LIN {X -192.412,Y -0.639,Z -49.375,A 0.015,B 0.000,C 180.000} C_DIS
LIN {X -191.183,Y 5.850,Z -49.619,A 0.015,B 0.000,C 180.000} C_DIS
LIN {X -196.636,Y 9.577,Z -49.863,A 0.015,B 0.000,C 180.000} C_DIS
LIN {X -202.235,Y 6.074,Z -50.107,A 0.015,B 0.000,C 180.000} C_DIS
LIN {X -201.270,Y -0.459,Z -50.351,A 0.015,B 0.000,C 180.000} C_DIS
LIN {X -194.897,Y -2.193,Z -50.595,A 0.015,B 0.000,C -180.000} C_DIS
LIN {X -190.755,Y 2.951,Z -50.839,A 0.015,B 0.000,C 180.000} C_DIS
LIN {X -193.808,Y 8.807,Z -51.083,A 0.015,B 0.000,C 180.000} C_DIS
LIN {X -200.397,Y 8.357,Z -51.327,A 0.015,B 0.000,C -180.000} C_DIS
LIN {X -202.624,Y 2.139,Z -51.571,A 0.015,B 0.000,C -180.000} C_DIS
LIN {X -197.821,Y -2.393,Z -51.815,A 0.015,B 0.000,C 180.000} C_DIS
LIN {X -191.743,Y 0.192,Z -52.060,A 0.015,B 0.000,C -180.000} C_DIS
LIN {X -191.677,Y 6.796,Z -52.304,A 0.015,B 0.000,C 180.000} C_DIS
LIN {X -197.700,Y 9.504,Z -52.548,A 0.015,B -0.000,C 180.000} C_DIS
LIN {X -202.595,Y 5.070,Z -52.792,A 0.015,B 0.000,C 180.000} C_DIS
LIN {X -200.494,Y -1.191,Z -53.036,A 0.015,B 0.000,C 180.000} C_DIS
LIN {X -193.915,Y -1.775,Z -53.280,A 0.015,B 0.000,C -180.000} C_DIS
LIN {X -190.744,Y 4.018,Z -53.524,A 0.015,B -0.000,C 180.000} C_DIS
LIN {X -194.781,Y 9.245,Z -53.768,A 0.015,B 0.000,C -180.000} C_DIS
LIN {X -201.188,Y 7.640,Z -54.012,A 0.015,B 0.000,C -180.000} C_DIS
LIN {X -202.285,Y 1.128,Z -54.256,A 0.015,B -0.000,C 180.000} C_DIS
LIN {X -196.758,Y -2.487,Z -54.500,A 0.015,B 0.000,C 180.000} C_DIS
LIN {X -193.305,Y -2.487,Z -54.500,A 0.015,B 0.000,C 180.000} C_DIS
CIRC {X -191.945,Y -1.389,Z -54.500,A 0.015,B 0.000,C 180.000},{X -192.732,Y 0.173,Z -54.500,A 0.015,B 0.000,C 180.000} C_DIS
CIRC {X -193.494,Y 0.521,Z -54.500,A 0.015,B 0.000,C -180.000},{X -194.253,Y 0.875,Z -54.500,A 0.015,B -0.000,C -180.000} C_DIS
CIRC {X -195.005,Y 1.244,Z -54.500,A 0.015,B 0.000,C 180.000},{X -195.745,Y 1.635,Z -54.500,A 0.015,B 0.000,C 180.000} C_DIS
CIRC {X -196.775,Y 1.894,Z -54.500,A 0.015,B 0.000,C -180.000},{X -197.801,Y 1.619,Z -54.500,A 0.015,B 0.000,C 180.000} C_DIS
CIRC {X -198.507,Y 1.231,Z -54.500,A 0.015,B 0.000,C -180.000},{X -199.224,Y 0.863,Z -54.500,A 0.015,B 0.000,C 180.000} C_DIS
CIRC {X -199.949,Y 0.511,Z -54.500,A 0.015,B 0.000,C 180.000},{X -200.680,Y 0.172,Z -54.500,A 0.015,B 0.000,C -180.000} C_DIS
CIRC {X -201.468,Y -1.389,Z -54.500,A 0.015,B -0.000,C 180.000},{X -200.108,Y -2.487,Z -54.500,A 0.015,B 0.000,C 180.000} C_DIS
LIN {X -196.758,Y -2.487,Z -54.500,A 0.015,B 0.000,C 180.000} C_DIS
CIRC {X -194.703,Y -3.109,Z -54.500,A 0.015,B -0.000,C 180.000},{X -193.339,Y -4.767,Z -54.500,A 0.015,B 0.000,C -180.000} C_DIS
CIRC {X -191.974,Y -6.424,Z -54.500,A 0.015,B 0.000,C -180.000},{X -189.919,Y -7.047,Z -54.500,A 0.015,B 0.000,C -180.000} C_DIS
LIN {X -172.141,Y -7.047,Z -54.500,A 0.015,B 0.000,C 180.000} C_DIS
CIRC {X -170.781,Y -5.948,Z -54.500,A 0.015,B -0.000,C -180.000},{X -171.568,Y -4.387,Z -54.500,A 0.015,B -0.000,C 180.000} C_DIS
CIRC {X -177.271,Y -1.878,Z -54.500,A 0.015,B -0.000,C -180.000},{X -183.023,Y 0.518,Z -54.500,A 0.015,B 0.000,C 180.000} C_DIS
CIRC {X -188.715,Y 3.061,Z -54.500,A 0.015,B 0.000,C 180.000},{X -194.211,Y 6.003,Z -54.500,A 0.015,B 0.000,C 180.000} C_DIS
CIRC {X -196.812,Y 6.694,Z -54.500,A 0.015,B 0.000,C -180.000},{X -199.402,Y 5.963,Z -54.500,A 0.015,B -0.000,C -180.000} C_DIS
CIRC {X -204.829,Y 2.985,Z -54.500,A 0.015,B 0.000,C -180.000},{X -210.480,Y 0.455,Z -54.500,A 0.015,B 0.000,C 180.000} C_DIS
CIRC {X -216.198,Y -1.904,Z -54.500,A 0.015,B 0.000,C 180.000},{X -221.864,Y -4.387,Z -54.500,A 0.015,B -0.000,C 180.000} C_DIS
CIRC {X -222.652,Y -5.948,Z -54.500,A 0.015,B 0.000,C -180.000},{X -221.292,Y -7.047,Z -54.500,A 0.015,B 0.000,C 180.000} C_DIS
LIN {X -189.919,Y -7.047,Z -54.500,A 0.015,B 0.000,C -180.000} C_DIS
CIRC {X -187.085,Y -7.904,Z -54.500,A 0.015,B 0.000,C 180.000},{X -185.204,Y -10.190,Z -54.500,A 0.015,B -0.000,C -180.000} C_DIS
CIRC {X -183.322,Y -12.476,Z -54.500,A 0.015,B 0.000,C -180.000},{X -180.488,Y -13.334,Z -54.500,A 0.015,B 0.000,C 180.000} C_DIS
LIN {X -142.956,Y -13.334,Z -54.500,A 0.015,B 0.000,C 180.000} C_DIS
CIRC {X -141.596,Y -12.235,Z -54.500,A 0.015,B 0.000,C 180.000},{X -142.383,Y -10.674,Z -54.500,A 0.015,B 0.000,C 180.000} C_DIS
LIN {X -189.172,Y 10.284,Z -54.500,A 0.015,B -0.000,C 180.000} C_DIS
CIRC {X -190.364,Y 10.896,Z -54.500,A 0.015,B 0.000,C 180.000},{X -191.488,Y 11.625,Z -54.500,A 0.015,B 0.000,C -180.000} C_DIS
CIRC {X -192.572,Y 12.410,Z -54.500,A 0.015,B 0.000,C 180.000},{X -193.651,Y 13.201,Z -54.500,A 0.015,B 0.000,C 180.000} C_DIS
CIRC {X -196.677,Y 14.214,Z -54.500,A 0.015,B 0.000,C 180.000},{X -199.724,Y 13.268,Z -54.500,A 0.015,B 0.000,C -180.000} C_DIS
CIRC {X -200.958,Y 12.395,Z -54.500,A 0.015,B 0.000,C 180.000},{X -202.187,Y 11.516,Z -54.500,A 0.015,B 0.000,C -180.000} C_DIS
CIRC {X -203.459,Y 10.695,Z -54.500,A 0.015,B 0.000,C -180.000},{X -204.805,Y 10.005,Z -54.500,A 0.015,B 0.000,C -180.000} C_DIS
LIN {X -251.078,Y -10.675,Z -54.500,A 0.015,B 0.000,C -180.000} C_DIS
CIRC {X -251.866,Y -12.235,Z -54.500,A 0.015,B 0.000,C 180.000},{X -250.505,Y -13.334,Z -54.500,A 0.015,B 0.000,C -180.000} C_DIS
LIN {X -180.488,Y -13.334,Z -54.500,A 0.015,B 0.000,C 180.000} C_DIS
CIRC {X -177.654,Y -14.192,Z -54.500,A 0.015,B 0.000,C 180.000},{X -175.772,Y -16.478,Z -54.500,A 0.015,B 0.000,C -180.000} C_DIS
CIRC {X -173.891,Y -18.763,Z -54.500,A 0.015,B -0.000,C -180.000},{X -171.057,Y -19.621,Z -54.500,A 0.015,B 0.000,C 180.000} C_DIS
LIN {X -113.771,Y -19.621,Z -54.500,A 0.015,B 0.000,C 180.000} C_DIS
CIRC {X -112.410,Y -18.523,Z -54.500,A 0.015,B 0.000,C 180.000},{X -113.198,Y -16.962,Z -54.500,A 0.015,B 0.000,C 180.000} C_DIS
LIN {X -186.653,Y 15.858,Z -54.500,A 0.015,B 0.000,C -180.000} C_DIS
CIRC {X -189.034,Y 17.198,Z -54.500,A 0.015,B 0.000,C 180.000},{X -191.144,Y 18.934,Z -54.500,A 0.015,B 0.000,C -180.000} C_DIS
CIRC {X -193.015,Y 20.912,Z -54.500,A 0.015,B 0.000,C -180.000},{X -194.736,Y 23.023,Z -54.500,A 0.015,B 0.000,C 180.000} C_DIS
CIRC {X -196.819,Y 24.035,Z -54.500,A 0.015,B 0.000,C 180.000},{X -198.863,Y 22.946,Z -54.500,A 0.015,B 0.000,C 180.000} C_DIS
CIRC {X -199.889,Y 21.563,Z -54.500,A 0.015,B -0.000,C 180.000},{X -200.992,Y 20.240,Z -54.500,A 0.015,B 0.000,C -180.000} C_DIS
CIRC {X -202.216,Y 19.026,Z -54.500,A 0.015,B 0.000,C 180.000},{X -203.590,Y 17.983,Z -54.500,A 0.015,B 0.000,C 180.000} C_DIS
CIRC {X -204.508,Y 17.359,Z -54.500,A 0.015,B -0.000,C -180.000},{X -205.410,Y 16.710,Z -54.500,A 0.015,B 0.000,C 180.000} C_DIS
CIRC {X -206.337,Y 16.098,Z -54.500,A 0.015,B 0.000,C -180.000},{X -207.325,Y 15.587,Z -54.500,A 0.015,B 0.000,C 180.000} C_DIS
LIN {X -280.291,Y -16.962,Z -54.500,A 0.015,B 0.000,C -180.000} C_DIS
CIRC {X -281.079,Y -18.523,Z -54.500,A 0.015,B 0.000,C 180.000},{X -279.719,Y -19.621,Z -54.500,A 0.015,B -0.000,C -180.000} C_DIS
LIN {X -171.057,Y -19.621,Z -54.500,A 0.015,B -0.000,C 180.000} C_DIS
LIN {X -170.448,Y -19.466,Z -54.330,A 0.015,B 0.000,C 180.000} C_DIS
LIN {X -170.089,Y -19.174,Z -53.865,A 0.015,B 0.000,C 180.000} C_DIS
LIN {X -169.988,Y -19.038,Z -53.230,A 0.015,B 0.000,C 180.000} C_DIS
$VEL.CP = 1.00000
LIN {X -169.988,Y -19.038,Z 11.000,A 0.015,B 0.000,C -180.000} C_DIS
$VEL.CP = 1.00000
LIN {X -57.220,Y 262.988,Z 11.000,A 0.015,B -0.000,C -180.000} C_DIS
$VEL.CP = 1.00000
LIN {X -57.220,Y 262.988,Z -32.731,A 0.015,B 0.000,C 180.000} C_DIS
$VEL.CP = 0.10000
LIN {X -57.218,Y 263.151,Z -33.353,A 0.015,B 0.000,C 180.000} C_DIS
LIN {X -57.234,Y 263.597,Z -33.816,A 0.015,B 0.000,C -180.000} C_DIS
LIN {X -57.310,Y 264.209,Z -34.000,A 0.015,B 0.000,C -180.000} C_DIS
LIN {X -61.835,Y 269.020,Z -34.244,A 0.015,B 0.000,C 180.000} C_DIS
LIN {X -68.056,Y 266.803,Z -34.488,A 0.015,B -0.000,C -180.000} C_DIS
LIN {X -68.517,Y 260.215,Z -34.732,A 0.015,B -0.000,C -180.000} C_DIS
LIN {X -62.666,Y 257.152,Z -34.976,A 0.015,B 0.000,C 180.000} C_DIS
LIN {X -57.515,Y 261.285,Z -35.220,A 0.015,B 0.000,C -180.000} C_DIS
LIN {X -59.238,Y 267.661,Z -35.464,A 0.015,B 0.000,C -180.000} C_DIS
LIN {X -65.770,Y 268.637,Z -35.708,A 0.015,B 0.000,C -180.000} C_DIS
LIN {X -69.282,Y 263.044,Z -35.952,A 0.015,B 0.000,C -180.000} C_DIS
LIN {X -65.565,Y 257.585,Z -36.196,A 0.015,B -0.000,C 180.000} C_DIS
LIN {X -59.074,Y 258.803,Z -36.440,A 0.015,B 0.000,C -180.000} C_DIS
LIN {X -57.589,Y 265.238,Z -36.685,A 0.015,B 0.000,C -180.000} C_DIS
LIN {X -62.890,Y 269.178,Z -36.929,A 0.015,B -0.000,C 180.000} C_DIS
LIN {X -68.623,Y 265.900,Z -37.173,A 0.015,B -0.000,C 180.000} C_DIS
LIN {X -67.917,Y 259.333,Z -37.417,A 0.015,B 0.000,C 180.000} C_DIS
LIN {X -61.618,Y 257.348,Z -37.661,A 0.015,B 0.000,C -180.000} C_DIS
LIN {X -57.275,Y 262.324,Z -37.905,A 0.015,B 0.000,C -180.000} C_DIS
LIN {X -60.094,Y 268.297,Z -38.149,A 0.015,B 0.000,C 180.000} C_DIS
LIN {X -66.696,Y 268.108,Z -38.393,A 0.015,B 0.000,C 180.000} C_DIS
LIN {X -69.168,Y 261.983,Z -38.637,A 0.015,B 0.000,C -180.000} C_DIS
LIN {X -64.547,Y 257.264,Z -38.881,A 0.015,B 0.000,C -180.000} C_DIS
LIN {X -58.372,Y 259.607,Z -39.125,A 0.015,B 0.000,C 180.000} C_DIS
LIN {X -58.044,Y 266.203,Z -39.369,A 0.015,B 0.000,C 180.000} C_DIS
LIN {X -63.956,Y 269.147,Z -39.613,A 0.015,B 0.000,C -180.000} C_DIS
LIN {X -69.022,Y 264.910,Z -39.857,A 0.015,B 0.000,C 180.000} C_DIS
LIN {X -67.171,Y 258.571,Z -40.101,A 0.015,B -0.000,C 180.000} C_DIS
LIN {X -60.621,Y 257.727,Z -40.345,A 0.015,B 0.000,C -180.000} C_DIS
LIN {X -57.222,Y 263.390,Z -40.589,A 0.015,B 0.000,C 180.000} C_DIS
LIN {X -61.049,Y 268.772,Z -40.833,A 0.015,B 0.000,C -180.000} C_DIS
LIN {X -67.514,Y 267.423,Z -41.077,A 0.015,B 0.000,C -180.000} C_DIS
LIN {X -68.869,Y 260.959,Z -41.321,A 0.015,B 0.000,C -180.000} C_DIS
LIN {X -63.489,Y 257.128,Z -41.565,A 0.015,B 0.000,C 180.000} C_DIS
LIN {X -57.824,Y 260.521,Z -41.810,A 0.015,B 0.000,C 180.000} C_DIS
LIN {X -58.662,Y 267.072,Z -42.054,A 0.015,B 0.000,C 180.000} C_DIS
LIN {X -65.000,Y 268.929,Z -42.298,A 0.015,B 0.000,C -180.000} C_DIS
LIN {X -69.241,Y 263.866,Z -42.542,A 0.015,B 0.000,C 180.000} C_DIS
LIN {X -66.302,Y 257.952,Z -42.786,A 0.015,B 0.000,C 180.000} C_DIS
LIN {X -59.705,Y 258.275,Z -43.030,A 0.015,B 0.000,C 180.000} C_DIS
LIN {X -57.358,Y 264.448,Z -43.274,A 0.015,B 0.000,C -180.000} C_DIS
LIN {X -62.073,Y 269.072,Z -43.518,A 0.015,B 0.000,C -180.000} C_DIS
LIN {X -68.199,Y 266.606,Z -43.762,A 0.015,B 0.000,C -180.000} C_DIS
LIN {X -68.394,Y 260.004,Z -44.006,A 0.015,B 0.000,C 180.000} C_DIS
LIN {X -62.424,Y 257.180,Z -44.250,A 0.015,B 0.000,C -180.000} C_DIS
LIN {X -57.444,Y 261.518,Z -44.494,A 0.015,B 0.000,C 180.000} C_DIS
LIN {X -59.424,Y 267.819,Z -44.738,A 0.015,B 0.000,C -180.000} C_DIS
LIN {X -65.989,Y 268.531,Z -44.982,A 0.015,B 0.000,C -180.000} C_DIS
LIN {X -69.272,Y 262.800,Z -45.226,A 0.015,B 0.000,C 180.000} C_DIS
LIN {X -65.338,Y 257.496,Z -45.470,A 0.015,B -0.000,C 180.000} C_DIS
LIN {X -58.901,Y 258.976,Z -45.714,A 0.015,B -0.000,C 180.000} C_DIS
LIN {X -57.678,Y 265.465,Z -45.958,A 0.015,B 0.000,C -180.000} C_DIS
LIN {X -63.133,Y 269.187,Z -46.202,A 0.015,B -0.000,C 180.000} C_DIS
LIN {X -68.729,Y 265.680,Z -46.446,A 0.015,B 0.000,C 180.000} C_DIS
LIN {X -67.759,Y 259.148,Z -46.690,A 0.015,B 0.000,C -180.000} C_DIS
LIN {X -61.384,Y 257.419,Z -46.935,A 0.015,B -0.000,C -180.000} C_DIS
LIN {X -57.247,Y 262.567,Z -47.179,A 0.015,B 0.000,C 180.000} C_DIS
LIN {X -60.305,Y 268.420,Z -47.423,A 0.015,B 0.000,C -180.000} C_DIS
LIN {X -66.893,Y 267.964,Z -47.667,A 0.015,B 0.000,C -180.000} C_DIS
LIN {X -69.116,Y 261.745,Z -47.911,A 0.015,B 0.000,C 180.000} C_DIS
LIN {X -64.308,Y 257.217,Z -48.155,A 0.015,B -0.000,C 180.000} C_DIS
LIN {X -58.233,Y 259.807,Z -48.399,A 0.015,B -0.000,C 180.000} C_DIS
LIN {X -58.171,Y 266.411,Z -48.643,A 0.015,B 0.000,C 180.000} C_DIS
LIN {X -64.197,Y 269.114,Z -48.887,A 0.015,B 0.000,C -180.000} C_DIS
LIN {X -69.088,Y 264.676,Z -49.131,A 0.015,B -0.000,C -180.000} C_DIS
LIN {X -66.982,Y 258.416,Z -49.375,A 0.015,B 0.000,C 180.000} C_DIS
LIN {X -60.403,Y 257.838,Z -49.619,A 0.015,B 0.000,C 180.000} C_DIS
LIN {X -57.237,Y 263.633,Z -49.863,A 0.015,B 0.000,C 180.000} C_DIS
LIN {X -61.278,Y 268.857,Z -50.107,A 0.015,B 0.000,C 180.000} C_DIS
LIN {X -67.683,Y 267.247,Z -50.351,A 0.015,B 0.000,C -180.000} C_DIS
LIN {X -68.775,Y 260.734,Z -50.595,A 0.015,B 0.000,C 180.000} C_DIS
LIN {X -63.246,Y 257.123,Z -50.839,A 0.015,B 0.000,C -180.000} C_DIS
LIN {X -57.721,Y 260.743,Z -51.083,A 0.015,B 0.000,C -180.000} C_DIS
LIN {X -58.824,Y 267.255,Z -51.327,A 0.015,B -0.000,C 180.000} C_DIS
LIN {X -65.232,Y 268.854,Z -51.571,A 0.015,B 0.000,C -180.000} C_DIS
LIN {X -69.265,Y 263.624,Z -51.815,A 0.015,B 0.000,C 180.000} C_DIS
LIN {X -66.089,Y 257.833,Z -52.060,A 0.015,B 0.000,C 180.000} C_DIS
LIN {X -59.511,Y 258.422,Z -52.304,A 0.015,B 0.000,C 180.000} C_DIS
LIN {X -57.415,Y 264.685,Z -52.548,A 0.015,B 0.000,C -180.000} C_DIS
LIN {X -62.313,Y 269.115,Z -52.792,A 0.015,B 0.000,C -180.000} C_DIS
LIN {X -68.335,Y 266.403,Z -53.036,A 0.015,B -0.000,C 180.000} C_DIS
LIN {X -68.262,Y 259.799,Z -53.280,A 0.015,B 0.000,C 180.000} C_DIS
LIN {X -62.183,Y 257.219,Z -53.524,A 0.015,B 0.000,C 180.000} C_DIS
LIN {X -57.383,Y 261.754,Z -53.768,A 0.015,B -0.000,C -180.000} C_DIS
LIN {X -59.615,Y 267.970,Z -54.012,A 0.015,B 0.000,C 180.000} C_DIS
LIN {X -66.204,Y 268.416,Z -54.256,A 0.015,B 0.000,C -180.000} C_DIS
LIN {X -69.253,Y 262.557,Z -54.500,A 0.015,B 0.000,C 180.000} C_DIS
LIN {X -65.146,Y 221.387,Z -54.500,A 0.015,B 0.000,C 180.000} C_DIS
CIRC {X -63.949,Y 220.356,Z -54.500,A 0.015,B 0.000,C -180.000},{X -62.860,Y 221.500,Z -54.500,A 0.015,B 0.000,C 180.000} C_DIS
LIN {X -62.861,Y 263.241,Z -54.500,A 0.015,B 0.000,C 180.000} C_DIS
CIRC {X -63.692,Y 265.248,Z -54.500,A 0.015,B -0.000,C -180.000},{X -65.699,Y 266.079,Z -54.500,A 0.015,B 0.000,C -180.000} C_DIS
LIN {X -66.469,Y 266.079,Z -54.500,A 0.015,B 0.000,C 180.000} C_DIS
CIRC {X -68.573,Y 265.145,Z -54.500,A 0.015,B 0.000,C 180.000},{X -69.293,Y 262.959,Z -54.500,A 0.015,B -0.000,C -180.000} C_DIS
LIN {X -69.253,Y 262.557,Z -54.500,A 0.015,B 0.000,C 180.000} C_DIS
CIRC {X -69.735,Y 260.112,Z -54.500,A 0.015,B 0.000,C -180.000},{X -71.492,Y 258.345,Z -54.500,A 0.015,B 0.000,C 180.000} C_DIS
CIRC {X -73.249,Y 256.577,Z -54.500,A 0.015,B 0.000,C -180.000},{X -73.731,Y 254.132,Z -54.500,A 0.015,B -0.000,C -180.000} C_DIS
LIN {X -66.932,Y 185.980,Z -54.500,A 0.015,B 0.000,C -180.000} C_DIS
CIRC {X -66.441,Y 184.456,Z -54.500,A 0.015,B 0.000,C 180.000},{X -65.366,Y 183.268,Z -54.500,A 0.015,B 0.000,C 180.000} C_DIS
LIN {X -60.809,Y 179.993,Z -54.500,A 0.015,B 0.000,C -180.000} C_DIS
CIRC {X -58.680,Y 179.834,Z -54.500,A 0.015,B 0.000,C -180.000},{X -57.566,Y 181.656,Z -54.500,A 0.015,B -0.000,C -180.000} C_DIS
LIN {X -57.569,Y 267.519,Z -54.500,A 0.015,B -0.000,C -180.000} C_DIS
CIRC {X -58.697,Y 270.243,Z -54.500,A 0.015,B 0.000,C 180.000},{X -61.422,Y 271.372,Z -54.500,A 0.015,B 0.000,C 180.000} C_DIS
LIN {X -71.668,Y 271.371,Z -54.500,A 0.015,B 0.000,C 180.000} C_DIS
CIRC {X -74.207,Y 270.245,Z -54.500,A 0.015,B 0.000,C 180.000},{X -75.076,Y 267.607,Z -54.500,A 0.015,B -0.000,C -180.000} C_DIS
LIN {X -73.731,Y 254.132,Z -54.500,A 0.015,B 0.000,C 180.000} C_DIS
CIRC {X -74.442,Y 250.524,Z -54.500,A 0.015,B 0.000,C -180.000},{X -77.035,Y 247.916,Z -54.500,A 0.015,B 0.000,C -180.000} C_DIS
CIRC {X -79.628,Y 245.308,Z -54.500,A 0.015,B 0.000,C -180.000},{X -80.339,Y 241.700,Z -54.500,A 0.015,B 0.000,C -180.000} C_DIS
LIN {X -74.727,Y 185.448,Z -54.500,A 0.015,B -0.000,C -180.000} C_DIS
CIRC {X -73.159,Y 180.577,Z -54.500,A 0.015,B 0.000,C 180.000},{X -69.725,Y 176.784,Z -54.500,A 0.015,B -0.000,C -180.000} C_DIS
LIN {X -52.999,Y 164.764,Z -54.500,A 0.015,B 0.000,C -180.000} C_DIS
CIRC {X -50.869,Y 164.604,Z -54.500,A 0.015,B -0.000,C -180.000},{X -49.756,Y 166.427,Z -54.500,A 0.015,B -0.000,C -180.000} C_DIS
LIN {X -49.759,Y 275.329,Z -54.500,A 0.015,B 0.000,C -180.000} C_DIS
CIRC {X -50.888,Y 278.053,Z -54.500,A 0.015,B 0.000,C 180.000},{X -53.612,Y 279.182,Z -54.500,A 0.015,B 0.000,C -180.000} C_DIS
LIN {X -80.296,Y 279.181,Z -54.500,A 0.015,B 0.000,C -180.000} C_DIS
CIRC {X -82.835,Y 278.055,Z -54.500,A 0.015,B 0.000,C 180.000},{X -83.703,Y 275.416,Z -54.500,A 0.015,B 0.000,C -180.000} C_DIS
LIN {X -80.339,Y 241.700,Z -54.500,A 0.015,B 0.000,C -180.000} C_DIS
CIRC {X -81.050,Y 238.092,Z -54.500,A 0.015,B -0.000,C 180.000},{X -83.644,Y 235.484,Z -54.500,A 0.015,B 0.000,C 180.000} C_DIS
CIRC {X -86.237,Y 232.876,Z -54.500,A 0.015,B 0.000,C 180.000},{X -86.948,Y 229.268,Z -54.500,A 0.015,B 0.000,C 180.000} C_DIS
LIN {X -82.181,Y 181.488,Z -54.500,A 0.015,B 0.000,C -180.000} C_DIS
CIRC {X -80.519,Y 176.328,Z -54.500,A 0.015,B -0.000,C -180.000},{X -76.882,Y 172.310,Z -54.500,A 0.015,B -0.000,C 180.000} C_DIS
LIN {X -45.189,Y 149.534,Z -54.500,A 0.015,B 0.000,C -180.000} C_DIS
CIRC {X -43.059,Y 149.375,Z -54.500,A 0.015,B -0.000,C 180.000},{X -41.946,Y 151.197,Z -54.500,A 0.015,B 0.000,C -180.000} C_DIS
LIN {X -41.949,Y 283.139,Z -54.500,A 0.015,B 0.000,C 180.000} C_DIS
CIRC {X -43.078,Y 285.863,Z -54.500,A 0.015,B 0.000,C -180.000},{X -45.802,Y 286.992,Z -54.500,A 0.015,B -0.000,C 180.000} C_DIS
LIN {X -88.923,Y 286.991,Z -54.500,A 0.015,B -0.000,C 180.000} C_DIS
CIRC {X -91.462,Y 285.864,Z -54.500,A 0.015,B 0.000,C 180.000},{X -92.331,Y 283.226,Z -54.500,A 0.015,B -0.000,C 180.000} C_DIS
LIN {X -86.948,Y 229.268,Z -54.500,A 0.015,B -0.000,C -180.000} C_DIS
CIRC {X -87.659,Y 225.660,Z -54.500,A 0.015,B 0.000,C -180.000},{X -90.252,Y 223.052,Z -54.500,A 0.015,B 0.000,C -180.000} C_DIS
CIRC {X -92.845,Y 220.444,Z -54.500,A 0.015,B 0.000,C 180.000},{X -93.556,Y 216.836,Z -54.500,A 0.015,B 0.000,C 180.000} C_DIS
LIN {X -89.602,Y 177.203,Z -54.500,A 0.015,B 0.000,C 180.000} C_DIS
CIRC {X -87.941,Y 172.044,Z -54.500,A 0.015,B 0.000,C 180.000},{X -84.303,Y 168.025,Z -54.500,A 0.015,B -0.000,C 180.000} C_DIS
LIN {X -37.378,Y 134.304,Z -54.500,A 0.015,B 0.000,C -180.000} C_DIS
CIRC {X -35.249,Y 134.145,Z -54.500,A 0.015,B 0.000,C 180.000},{X -34.136,Y 135.967,Z -54.500,A 0.015,B -0.000,C -180.000} C_DIS
LIN {X -34.140,Y 290.949,Z -54.500,A 0.015,B 0.000,C -180.000} C_DIS
CIRC {X -35.268,Y 293.673,Z -54.500,A 0.015,B 0.000,C 180.000},{X -37.993,Y 294.802,Z -54.500,A 0.015,B 0.000,C 180.000} C_DIS
LIN {X -97.551,Y 294.800,Z -54.500,A 0.015,B -0.000,C 180.000} C_DIS
CIRC {X -100.090,Y 293.674,Z -54.500,A 0.015,B -0.000,C 180.000},{X -100.959,Y 291.036,Z -54.500,A 0.015,B 0.000,C 180.000} C_DIS
LIN {X -93.556,Y 216.836,Z -54.500,A 0.015,B 0.000,C -180.000} C_DIS
CIRC {X -94.268,Y 213.222,Z -54.500,A 0.015,B 0.000,C -180.000},{X -96.864,Y 210.610,Z -54.500,A 0.015,B 0.000,C -180.000} C_DIS
CIRC {X -99.460,Y 207.998,Z -54.500,A 0.015,B 0.000,C -180.000},{X -100.171,Y 204.384,Z -54.500,A 0.015,B 0.000,C -180.000} C_DIS
LIN {X -97.023,Y 172.919,Z -54.500,A 0.015,B 0.000,C -180.000} C_DIS
CIRC {X -95.362,Y 167.760,Z -54.500,A 0.015,B 0.000,C -180.000},{X -91.724,Y 163.741,Z -54.500,A 0.015,B 0.000,C 180.000} C_DIS
LIN {X -29.568,Y 119.075,Z -54.500,A 0.015,B 0.000,C 180.000} C_DIS
CIRC {X -27.439,Y 118.915,Z -54.500,A 0.015,B 0.000,C -180.000},{X -26.325,Y 120.738,Z -54.500,A 0.015,B 0.000,C -180.000} C_DIS
LIN {X -26.330,Y 298.759,Z -54.500,A 0.015,B 0.000,C 180.000} C_DIS
CIRC {X -27.459,Y 301.483,Z -54.500,A 0.015,B -0.000,C 180.000},{X -30.183,Y 302.612,Z -54.500,A 0.015,B 0.000,C -180.000} C_DIS
LIN {X -106.248,Y 302.610,Z -54.500,A 0.015,B 0.000,C 180.000} C_DIS
CIRC {X -108.774,Y 301.483,Z -54.500,A 0.015,B 0.000,C 180.000},{X -109.624,Y 298.852,Z -54.500,A 0.015,B 0.000,C 180.000} C_DIS
LIN {X -100.171,Y 204.384,Z -54.500,A 0.015,B -0.000,C 180.000} C_DIS
CIRC {X -100.875,Y 200.830,Z -54.500,A 0.015,B 0.000,C -180.000},{X -103.439,Y 198.271,Z -54.500,A 0.015,B 0.000,C 180.000} C_DIS
CIRC {X -105.996,Y 195.708,Z -54.500,A 0.015,B 0.000,C 180.000},{X -106.706,Y 192.157,Z -54.500,A 0.015,B 0.000,C -180.000} C_DIS
LIN {X -104.355,Y 167.741,Z -54.500,A 0.015,B 0.000,C -180.000} C_DIS
CIRC {X -102.950,Y 163.379,Z -54.500,A 0.015,B 0.000,C -180.000},{X -99.875,Y 159.981,Z -54.500,A 0.015,B -0.000,C -180.000} C_DIS
LIN {X -21.758,Y 103.845,Z -54.500,A 0.015,B -0.000,C 180.000} C_DIS
CIRC {X -19.628,Y 103.686,Z -54.500,A 0.015,B 0.000,C -180.000},{X -18.515,Y 105.508,Z -54.500,A 0.015,B 0.000,C 180.000} C_DIS
LIN {X -18.521,Y 306.569,Z -54.500,A 0.015,B 0.000,C 180.000} C_DIS
CIRC {X -19.649,Y 309.293,Z -54.500,A 0.015,B 0.000,C 180.000},{X -22.374,Y 310.422,Z -54.500,A 0.015,B 0.000,C -180.000} C_DIS
LIN {X -115.486,Y 310.419,Z -54.500,A 0.015,B -0.000,C 180.000} C_DIS
CIRC {X -117.830,Y 309.310,Z -54.500,A 0.015,B 0.000,C 180.000},{X -118.460,Y 306.795,Z -54.500,A 0.015,B -0.000,C -180.000} C_DIS
CIRC {X -117.276,Y 299.976,Z -54.500,A 0.015,B 0.000,C 180.000},{X -116.428,Y 293.107,Z -54.500,A 0.015,B 0.000,C -180.000} C_DIS
LIN {X -106.706,Y 192.157,Z -54.500,A 0.015,B -0.000,C -180.000} C_DIS
CIRC {X -107.419,Y 188.605,Z -54.500,A 0.015,B 0.000,C 180.000},{X -109.983,Y 186.044,Z -54.500,A 0.015,B 0.000,C -180.000} C_DIS
CIRC {X -112.546,Y 183.483,Z -54.500,A 0.015,B 0.000,C 180.000},{X -113.259,Y 179.930,Z -54.500,A 0.015,B 0.000,C 180.000} C_DIS
LIN {X -111.900,Y 165.827,Z -54.500,A 0.015,B -0.000,C 180.000} C_DIS
CIRC {X -111.841,Y 164.928,Z -54.500,A 0.015,B 0.000,C 180.000},{X -111.843,Y 164.026,Z -54.500,A 0.015,B 0.000,C 180.000} C_DIS
CIRC {X -111.879,Y 163.126,Z -54.500,A 0.015,B 0.000,C 180.000},{X -111.919,Y 162.226,Z -54.500,A 0.015,B 0.000,C 180.000} C_DIS
CIRC {X -111.054,Y 158.666,Z -54.500,A 0.015,B 0.000,C 180.000},{X -108.395,Y 156.145,Z -54.500,A 0.015,B 0.000,C 180.000} C_DIS
CIRC {X -107.575,Y 155.723,Z -54.500,A 0.015,B 0.000,C 180.000},{X -106.758,Y 155.295,Z -54.500,A 0.015,B 0.000,C 180.000} C_DIS
CIRC {X -105.958,Y 154.837,Z -54.500,A 0.015,B -0.000,C 180.000},{X -105.190,Y 154.325,Z -54.500,A 0.015,B 0.000,C 180.000} C_DIS
LIN {X -13.948,Y 88.615,Z -54.500,A 0.015,B 0.000,C -180.000} C_DIS
CIRC {X -11.818,Y 88.456,Z -54.500,A 0.015,B 0.000,C -180.000},{X -10.705,Y 90.278,Z -54.500,A 0.015,B 0.000,C 180.000} C_DIS
LIN {X -10.711,Y 314.379,Z -54.500,A 0.015,B 0.000,C 180.000} C_DIS
CIRC {X -11.840,Y 317.103,Z -54.500,A 0.015,B 0.000,C -180.000},{X -14.564,Y 318.232,Z -54.500,A 0.015,B -0.000,C 180.000} C_DIS
LIN {X -125.780,Y 318.229,Z -54.500,A 0.015,B -0.000,C -180.000} C_DIS
CIRC {X -127.944,Y 317.152,Z -54.500,A 0.015,B 0.000,C 180.000},{X -128.390,Y 314.776,Z -54.500,A 0.015,B -0.000,C 180.000} C_DIS
CIRC {X -125.771,Y 303.744,Z -54.500,A 0.015,B 0.000,C 180.000},{X -124.108,Y 292.528,Z -54.500,A 0.015,B -0.000,C 180.000} C_DIS
LIN {X -113.259,Y 179.930,Z -54.500,A 0.015,B -0.000,C 180.000} C_DIS
CIRC {X -113.965,Y 176.402,Z -54.500,A 0.015,B 0.000,C -180.000},{X -116.506,Y 173.856,Z -54.500,A 0.015,B -0.000,C -180.000} C_DIS
CIRC {X -119.051,Y 171.310,Z -54.500,A 0.015,B -0.000,C -180.000},{X -119.754,Y 167.781,Z -54.500,A 0.015,B -0.000,C 180.000} C_DIS
LIN {X -119.489,Y 165.070,Z -54.500,A 0.015,B 0.000,C 180.000} C_DIS
CIRC {X -119.427,Y 162.680,Z -54.500,A 0.015,B -0.000,C 180.000},{X -119.716,Y 160.306,Z -54.500,A 0.015,B -0.000,C -180.000} C_DIS
CIRC {X -120.244,Y 157.979,Z -54.500,A 0.015,B -0.000,C 180.000},{X -120.905,Y 155.686,Z -54.500,A 0.015,B 0.000,C -180.000} C_DIS
CIRC {X -120.644,Y 153.191,Z -54.500,A 0.015,B 0.000,C -180.000},{X -118.634,Y 151.690,Z -54.500,A 0.015,B 0.000,C 180.000} C_DIS
CIRC {X -116.926,Y 151.259,Z -54.500,A 0.015,B 0.000,C -180.000},{X -115.236,Y 150.764,Z -54.500,A 0.015,B 0.000,C -180.000} C_DIS
CIRC {X -113.576,Y 150.171,Z -54.500,A 0.015,B 0.000,C -180.000},{X -111.970,Y 149.447,Z -54.500,A 0.015,B 0.000,C 180.000} C_DIS
CIRC {X -111.373,Y 149.145,Z -54.500,A 0.015,B 0.000,C -180.000},{X -110.778,Y 148.837,Z -54.500,A 0.015,B 0.000,C 180.000} C_DIS
CIRC {X -110.196,Y 148.505,Z -54.500,A 0.015,B 0.000,C -180.000},{X -109.639,Y 148.134,Z -54.500,A 0.015,B 0.000,C 180.000} C_DIS
LIN {X -6.138,Y 73.385,Z -54.500,A 0.015,B 0.000,C -180.000} C_DIS
CIRC {X -4.008,Y 73.226,Z -54.500,A 0.015,B 0.000,C 180.000},{X -2.895,Y 75.048,Z -54.500,A 0.015,B -0.000,C -180.000} C_DIS
LIN {X -2.901,Y 322.189,Z -54.500,A 0.015,B -0.000,C -180.000} C_DIS
CIRC {X -4.030,Y 324.913,Z -54.500,A 0.015,B 0.000,C 180.000},{X -6.755,Y 326.042,Z -54.500,A 0.015,B 0.000,C -180.000} C_DIS
LIN {X -138.556,Y 326.038,Z -54.500,A 0.015,B 0.000,C -180.000} C_DIS
CIRC {X -140.500,Y 324.922,Z -54.500,A 0.015,B 0.000,C -180.000},{X -140.515,Y 322.681,Z -54.500,A 0.015,B 0.000,C 180.000} C_DIS
CIRC {X -138.936,Y 319.901,Z -54.500,A 0.015,B 0.000,C 180.000},{X -137.343,Y 317.129,Z -54.500,A 0.015,B 0.000,C -180.000} C_DIS
CIRC {X -135.984,Y 314.222,Z -54.500,A 0.015,B 0.000,C -180.000},{X -135.146,Y 311.124,Z -54.500,A 0.015,B 0.000,C -180.000} C_DIS
CIRC {X -134.260,Y 306.277,Z -54.500,A 0.015,B 0.000,C 180.000},{X -133.339,Y 301.438,Z -54.500,A 0.015,B 0.000,C 180.000} C_DIS
CIRC {X -132.503,Y 296.582,Z -54.500,A 0.015,B 0.000,C -180.000},{X -131.874,Y 291.695,Z -54.500,A 0.015,B 0.000,C 180.000} C_DIS
LIN {X -119.754,Y 167.781,Z -54.500,A 0.015,B 0.000,C -180.000} C_DIS
CIRC {X -120.533,Y 163.962,Z -54.500,A 0.015,B -0.000,C 180.000},{X -123.324,Y 161.243,Z -54.500,A 0.015,B 0.000,C 180.000} C_DIS
CIRC {X -126.370,Y 159.021,Z -54.500,A 0.015,B 0.000,C -180.000},{X -128.586,Y 155.970,Z -54.500,A 0.015,B 0.000,C -180.000} C_DIS
CIRC {X -129.163,Y 154.939,Z -54.500,A 0.015,B 0.000,C -180.000},{X -129.820,Y 153.956,Z -54.500,A 0.015,B 0.000,C 180.000} C_DIS
CIRC {X -133.257,Y 149.818,Z -54.500,A 0.015,B 0.000,C -180.000},{X -137.197,Y 146.156,Z -54.500,A 0.015,B 0.000,C 180.000} C_DIS
CIRC {X -137.836,Y 145.658,Z -54.500,A 0.015,B 0.000,C 180.000},{X -138.496,Y 145.188,Z -54.500,A 0.015,B -0.000,C -180.000} C_DIS
CIRC {X -139.174,Y 144.745,Z -54.500,A 0.015,B 0.000,C -180.000},{X -139.868,Y 144.327,Z -54.500,A 0.015,B 0.000,C 180.000} C_DIS
LIN {X -176.147,Y 123.347,Z -54.500,A 0.015,B 0.000,C -180.000} C_DIS
CIRC {X -181.598,Y 121.768,Z -54.500,A 0.015,B 0.000,C -180.000},{X -187.157,Y 122.914,Z -54.500,A 0.015,B 0.000,C 180.000} C_DIS
CIRC {X -191.634,Y 126.325,Z -54.500,A 0.015,B -0.000,C -180.000},{X -194.376,Y 131.240,Z -54.500,A 0.015,B 0.000,C -180.000} C_DIS
CIRC {X -194.694,Y 132.613,Z -54.500,A 0.015,B -0.000,C 180.000},{X -194.801,Y 134.019,Z -54.500,A 0.015,B 0.000,C -180.000} C_DIS
LIN {X -194.206,Y 259.887,Z -54.500,A 0.015,B -0.000,C 180.000} C_DIS
CIRC {X -194.825,Y 261.382,Z -54.500,A 0.015,B 0.000,C 180.000},{X -196.320,Y 262.002,Z -54.500,A 0.015,B 0.000,C 180.000} C_DIS
LIN {X -197.192,Y 262.002,Z -54.500,A 0.015,B 0.000,C -180.000} C_DIS
CIRC {X -198.687,Y 261.382,Z -54.500,A 0.015,B 0.000,C 180.000},{X -199.306,Y 259.887,Z -54.500,A 0.015,B 0.000,C -180.000} C_DIS
LIN {X -198.711,Y 134.015,Z -54.500,A 0.015,B -0.000,C 180.000} C_DIS
CIRC {X -200.100,Y 128.501,Z -54.500,A 0.015,B 0.000,C -180.000},{X -203.935,Y 124.303,Z -54.500,A 0.015,B 0.000,C 180.000} C_DIS
CIRC {X -209.158,Y 122.206,Z -54.500,A 0.015,B -0.000,C -180.000},{X -214.785,Y 122.333,Z -54.500,A 0.015,B 0.000,C 180.000} C_DIS
CIRC {X -215.493,Y 122.525,Z -54.500,A 0.015,B 0.000,C 180.000},{X -216.182,Y 122.776,Z -54.500,A 0.015,B 0.000,C 180.000} C_DIS
CIRC {X -216.850,Y 123.077,Z -54.500,A 0.015,B -0.000,C -180.000},{X -217.497,Y 123.423,Z -54.500,A 0.015,B -0.000,C 180.000} C_DIS
LIN {X -256.621,Y 146.379,Z -54.500,A 0.015,B -0.000,C -180.000} C_DIS
CIRC {X -260.341,Y 149.573,Z -54.500,A 0.015,B -0.000,C -180.000},{X -263.385,Y 153.418,Z -54.500,A 0.015,B -0.000,C -180.000} C_DIS
CIRC {X -265.525,Y 157.847,Z -54.500,A 0.015,B 0.000,C 180.000},{X -266.515,Y 162.665,Z -54.500,A 0.015,B 0.000,C -180.000} C_DIS
CIRC {X -266.544,Y 163.493,Z -54.500,A 0.015,B 0.000,C 180.000},{X -266.498,Y 164.321,Z -54.500,A 0.015,B 0.000,C -180.000} C_DIS
LIN {X -252.263,Y 304.023,Z -54.500,A 0.015,B -0.000,C -180.000} C_DIS
CIRC {X -250.701,Y 309.424,Z -54.500,A 0.015,B 0.000,C 180.000},{X -248.523,Y 314.608,Z -54.500,A 0.015,B 0.000,C -180.000} C_DIS
CIRC {X -245.977,Y 319.611,Z -54.500,A 0.015,B 0.000,C -180.000},{X -243.286,Y 324.538,Z -54.500,A 0.015,B 0.000,C 180.000} C_DIS
CIRC {X -242.051,Y 326.341,Z -54.500,A 0.015,B 0.000,C -180.000},{X -240.525,Y 327.906,Z -54.500,A 0.015,B 0.000,C -180.000} C_DIS
CIRC {X -238.890,Y 329.346,Z -54.500,A 0.015,B -0.000,C -180.000},{X -237.284,Y 330.817,Z -54.500,A 0.015,B 0.000,C 180.000} C_DIS
CIRC {X -236.851,Y 332.738,Z -54.500,A 0.015,B -0.000,C 180.000},{X -238.479,Y 333.846,Z -54.500,A 0.015,B 0.000,C 180.000} C_DIS
LIN {X -394.577,Y 333.842,Z -54.500,A 0.015,B 0.000,C 180.000} C_DIS
CIRC {X -397.301,Y 332.713,Z -54.500,A 0.015,B 0.000,C -180.000},{X -398.430,Y 329.989,Z -54.500,A 0.015,B -0.000,C -180.000} C_DIS
LIN {X -398.422,Y 58.290,Z -54.500,A 0.015,B -0.000,C -180.000} C_DIS
CIRC {X -397.314,Y 56.658,Z -54.500,A 0.015,B -0.000,C 180.000},{X -395.388,Y 57.085,Z -54.500,A 0.015,B -0.000,C -180.000} C_DIS
CIRC {X -393.075,Y 59.405,Z -54.500,A 0.015,B -0.000,C -180.000},{X -390.640,Y 61.595,Z -54.500,A 0.015,B -0.000,C -180.000} C_DIS
CIRC {X -388.103,Y 63.666,Z -54.500,A 0.015,B -0.000,C 180.000},{X -385.483,Y 65.631,Z -54.500,A 0.015,B 0.000,C 180.000} C_DIS
LIN {X -279.081,Y 142.208,Z -54.500,A 0.015,B -0.000,C -180.000} C_DIS
CIRC {X -274.197,Y 144.494,Z -54.500,A 0.015,B -0.000,C 180.000},{X -268.816,Y 144.860,Z -54.500,A 0.015,B -0.000,C 180.000} C_DIS
CIRC {X -263.590,Y 143.910,Z -54.500,A 0.015,B 0.000,C 180.000},{X -258.524,Y 142.314,Z -54.500,A 0.015,B 0.000,C 180.000} C_DIS
CIRC {X -257.668,Y 141.957,Z -54.500,A 0.015,B 0.000,C 180.000},{X -256.832,Y 141.554,Z -54.500,A 0.015,B -0.000,C 180.000} C_DIS
CIRC {X -256.012,Y 141.120,Z -54.500,A 0.015,B 0.000,C 180.000},{X -255.203,Y 140.667,Z -54.500,A 0.015,B -0.000,C 180.000} C_DIS
LIN {X -219.429,Y 120.082,Z -54.500,A 0.015,B 0.000,C -180.000} C_DIS
CIRC {X -215.282,Y 116.094,Z -54.500,A 0.015,B 0.000,C -180.000},{X -213.463,Y 110.636,Z -54.500,A 0.015,B 0.000,C -180.000} C_DIS
CIRC {X -214.201,Y 104.972,Z -54.500,A 0.015,B 0.000,C -180.000},{X -217.183,Y 100.101,Z -54.500,A 0.015,B 0.000,C 180.000} C_DIS
CIRC {X -218.178,Y 99.193,Z -54.500,A 0.015,B -0.000,C -180.000},{X -219.295,Y 98.439,Z -54.500,A 0.015,B 0.000,C -180.000} C_DIS
LIN {X -328.516,Y 36.081,Z -54.500,A 0.015,B 0.000,C -180.000} C_DIS
CIRC {X -329.501,Y 34.796,Z -54.500,A 0.015,B 0.000,C 180.000},{X -329.289,Y 33.191,Z -54.500,A 0.015,B -0.000,C -180.000} C_DIS
LIN {X -328.854,Y 32.438,Z -54.500,A 0.015,B 0.000,C 180.000} C_DIS
CIRC {X -327.570,Y 31.454,Z -54.500,A 0.015,B -0.000,C 180.000},{X -325.966,Y 31.666,Z -54.500,A 0.015,B -0.000,C -180.000} C_DIS
LIN {X -217.356,Y 95.076,Z -54.500,A 0.015,B -0.000,C -180.000} C_DIS
CIRC {X -211.853,Y 96.649,Z -54.500,A 0.015,B -0.000,C 180.000},{X -206.257,Y 95.448,Z -54.500,A 0.015,B 0.000,C 180.000} C_DIS
CIRC {X -201.784,Y 91.960,Z -54.500,A 0.015,B 0.000,C -180.000},{X -199.085,Y 86.971,Z -54.500,A 0.015,B 0.000,C 180.000} C_DIS
CIRC {X -198.795,Y 85.656,Z -54.500,A 0.015,B 0.000,C 180.000},{X -198.698,Y 84.312,Z -54.500,A 0.015,B -0.000,C -180.000} C_DIS
LIN {X -199.059,Y 38.427,Z -54.500,A 0.015,B 0.000,C 180.000} C_DIS
CIRC {X -200.026,Y 33.606,Z -54.500,A 0.015,B 0.000,C -180.000},{X -201.926,Y 29.071,Z -54.500,A 0.015,B 0.000,C -180.000} C_DIS
CIRC {X -204.786,Y 25.055,Z -54.500,A 0.015,B 0.000,C -180.000},{X -208.537,Y 21.856,Z -54.500,A 0.015,B 0.000,C -180.000} C_DIS
CIRC {X -209.171,Y 21.473,Z -54.500,A 0.015,B -0.000,C 180.000},{X -209.832,Y 21.142,Z -54.500,A 0.015,B 0.000,C -180.000} C_DIS
LIN {X -309.505,Y -23.249,Z -54.500,A 0.015,B -0.000,C 180.000} C_DIS
CIRC {X -310.293,Y -24.810,Z -54.500,A 0.015,B 0.000,C -180.000},{X -308.933,Y -25.909,Z -54.500,A 0.015,B -0.000,C 180.000} C_DIS
LIN {X -84.585,Y -25.909,Z -54.500,A 0.015,B 0.000,C 180.000} C_DIS
CIRC {X -83.225,Y -24.810,Z -54.500,A 0.015,B -0.000,C -180.000},{X -84.012,Y -23.249,Z -54.500,A 0.015,B 0.000,C 180.000} C_DIS
LIN {X -184.149,Y 21.400,Z -54.500,A 0.015,B -0.000,C 180.000} C_DIS
CIRC {X -188.274,Y 24.206,Z -54.500,A 0.015,B 0.000,C 180.000},{X -191.203,Y 28.245,Z -54.500,A 0.015,B 0.000,C -180.000} C_DIS
CIRC {X -193.071,Y 32.802,Z -54.500,A 0.015,B -0.000,C -180.000},{X -194.326,Y 37.565,Z -54.500,A 0.015,B 0.000,C -180.000} C_DIS
CIRC {X -194.665,Y 39.888,Z -54.500,A 0.015,B -0.000,C -180.000},{X -194.784,Y 42.234,Z -54.500,A 0.015,B 0.000,C -180.000} C_DIS
LIN {X -194.814,Y 84.319,Z -54.500,A 0.015,B 0.000,C -180.000} C_DIS
CIRC {X -193.075,Y 90.605,Z -54.500,A 0.015,B 0.000,C 180.000},{X -188.354,Y 95.105,Z -54.500,A 0.015,B 0.000,C -180.000} C_DIS
CIRC {X -182.042,Y 96.633,Z -54.500,A 0.015,B 0.000,C -180.000},{X -175.783,Y 94.898,Z -54.500,A 0.015,B -0.000,C 180.000} C_DIS
LIN {X -67.545,Y 31.669,Z -54.500,A 0.015,B 0.000,C -180.000} C_DIS
CIRC {X -65.941,Y 31.456,Z -54.500,A 0.015,B 0.000,C -180.000},{X -64.657,Y 32.440,Z -54.500,A 0.015,B -0.000,C 180.000} C_DIS
LIN {X -64.222,Y 33.191,Z -54.500,A 0.015,B -0.000,C -180.000} C_DIS
CIRC {X -64.011,Y 34.796,Z -54.500,A 0.015,B 0.000,C 180.000},{X -64.996,Y 36.081,Z -54.500,A 0.015,B 0.000,C -180.000} C_DIS
LIN {X -174.232,Y 98.448,Z -54.500,A 0.015,B -0.000,C -180.000} C_DIS
CIRC {X -178.431,Y 102.562,Z -54.500,A 0.015,B 0.000,C -180.000},{X -180.120,Y 108.193,Z -54.500,A 0.015,B 0.000,C 180.000} C_DIS
CIRC {X -179.122,Y 113.930,Z -54.500,A 0.015,B 0.000,C 180.000},{X -175.856,Y 118.750,Z -54.500,A 0.015,B -0.000,C -180.000} C_DIS
CIRC {X -175.001,Y 119.475,Z -54.500,A 0.015,B 0.000,C -180.000},{X -174.065,Y 120.092,Z -54.500,A 0.015,B 0.000,C 180.000} C_DIS
LIN {X -133.766,Y 142.826,Z -54.500,A 0.015,B 0.000,C -180.000} C_DIS
CIRC {X -129.253,Y 144.306,Z -54.500,A 0.015,B 0.000,C -180.000},{X -124.534,Y 144.854,Z -54.500,A 0.015,B 0.000,C -180.000} C_DIS
CIRC {X -119.800,Y 144.358,Z -54.500,A 0.015,B -0.000,C 180.000},{X -115.319,Y 142.752,Z -54.500,A 0.015,B -0.000,C 180.000} C_DIS
CIRC {X -114.672,Y 142.395,Z -54.500,A 0.015,B 0.000,C -180.000},{X -114.055,Y 141.988,Z -54.500,A 0.015,B 0.000,C 180.000} C_DIS
LIN {X -3.676,Y 62.273,Z -54.500,A 0.015,B -0.000,C -180.000} C_DIS
CIRC {X -2.226,Y 61.044,Z -54.500,A 0.015,B 0.000,C -180.000},{X -0.833,Y 59.752,Z -54.500,A 0.015,B -0.000,C -180.000} C_DIS
CIRC {X 0.529,Y 58.426,Z -54.500,A 0.015,B 0.000,C -180.000},{X 1.883,Y 57.094,Z -54.500,A 0.015,B 0.000,C 180.000} C_DIS
CIRC {X 3.821,Y 56.717,Z -54.500,A 0.015,B 0.000,C -180.000},{X 4.916,Y 58.360,Z -54.500,A 0.015,B -0.000,C 180.000} C_DIS
LIN {X 4.908,Y 329.999,Z -54.500,A 0.015,B 0.000,C 180.000} C_DIS
CIRC {X 3.780,Y 332.723,Z -54.500,A 0.015,B 0.000,C -180.000},{X 1.055,Y 333.852,Z -54.500,A 0.015,B -0.000,C 180.000} C_DIS
LIN {X -155.023,Y 333.848,Z -54.500,A 0.015,B 0.000,C 180.000} C_DIS
CIRC {X -156.652,Y 332.740,Z -54.500,A 0.015,B 0.000,C -180.000},{X -156.221,Y 330.817,Z -54.500,A 0.015,B 0.000,C 180.000} C_DIS
CIRC {X -154.617,Y 329.345,Z -54.500,A 0.015,B 0.000,C -180.000},{X -152.985,Y 327.905,Z -54.500,A 0.015,B 0.000,C -180.000} C_DIS
CIRC {X -151.460,Y 326.340,Z -54.500,A 0.015,B 0.000,C -180.000},{X -150.226,Y 324.538,Z -54.500,A 0.015,B -0.000,C -180.000} C_DIS
CIRC {X -147.842,Y 320.230,Z -54.500,A 0.015,B -0.000,C 180.000},{X -145.536,Y 315.880,Z -54.500,A 0.015,B 0.000,C -180.000} C_DIS
CIRC {X -143.482,Y 311.399,Z -54.500,A 0.015,B 0.000,C 180.000},{X -141.875,Y 306.740,Z -54.500,A 0.015,B -0.000,C 180.000} C_DIS
CIRC {X -140.944,Y 302.831,Z -54.500,A 0.015,B 0.000,C 180.000},{X -140.406,Y 298.850,Z -54.500,A 0.015,B 0.000,C 180.000} C_DIS
CIRC {X -140.045,Y 294.853,Z -54.500,A 0.015,B 0.000,C -180.000},{X -139.639,Y 290.861,Z -54.500,A 0.015,B 0.000,C 180.000} C_DIS
LIN {X -127.014,Y 164.319,Z -54.500,A 0.015,B 0.000,C -180.000} C_DIS
CIRC {X -127.200,Y 160.032,Z -54.500,A 0.015,B 0.000,C -180.000},{X -128.586,Y 155.970,Z -54.500,A 0.015,B 0.000,C 180.000} C_DIS
LIN {X -128.721,Y 155.356,Z -54.330,A 0.015,B 0.000,C 180.000} C_DIS
LIN {X -128.621,Y 154.905,Z -53.865,A 0.015,B -0.000,C -180.000} C_DIS
LIN {X -128.545,Y 154.753,Z -53.230,A 0.015,B 0.000,C -180.000} C_DIS
$VEL.CP = 1.00000
LIN {X -128.545,Y 154.753,Z 11.000,A 0.015,B 0.000,C 180.000} C_DIS
$VEL.CP = 1.00000
LIN {X 0.374,Y 325.785,Z 11.000,A 0.015,B 0.000,C -180.000} C_DIS
$VEL.CP = 0.10000
LIN {X 0.374,Y 325.785,Z -32.731,A 0.015,B 0.000,C 180.000} C_DIS
LIN {X 0.249,Y 325.889,Z -33.353,A 0.015,B 0.000,C 180.000} C_DIS
LIN {X -0.081,Y 326.190,Z -33.816,A 0.015,B 0.000,C 180.000} C_DIS
LIN {X -0.497,Y 326.645,Z -34.000,A 0.015,B 0.000,C 180.000} C_DIS
LIN {X -1.230,Y 333.208,Z -34.244,A 0.015,B -0.000,C -180.000} C_DIS
LIN {X 4.489,Y 336.510,Z -34.488,A 0.015,B 0.000,C -180.000} C_DIS
LIN {X 9.806,Y 332.593,Z -34.732,A 0.015,B 0.000,C 180.000} C_DIS
LIN {X 8.348,Y 326.152,Z -34.976,A 0.015,B 0.000,C -180.000} C_DIS
LIN {X 1.863,Y 324.906,Z -35.220,A 0.015,B 0.000,C 180.000} C_DIS
LIN {X -1.877,Y 330.350,Z -35.464,A 0.015,B 0.000,C 180.000} C_DIS
LIN {X 1.611,Y 335.958,Z -35.708,A 0.015,B -0.000,C 180.000} C_DIS
LIN {X 8.147,Y 335.009,Z -35.952,A 0.015,B 0.000,C -180.000} C_DIS
LIN {X 9.896,Y 328.640,Z -36.196,A 0.015,B 0.000,C -180.000} C_DIS
LIN {X 4.763,Y 324.485,Z -36.440,A 0.015,B 0.000,C -180.000} C_DIS
LIN {X -1.101,Y 327.524,Z -36.685,A 0.015,B 0.000,C -180.000} C_DIS
LIN {X -0.667,Y 334.114,Z -36.929,A 0.015,B -0.000,C 180.000} C_DIS
LIN {X 5.545,Y 336.357,Z -37.173,A 0.015,B 0.000,C -180.000} C_DIS
LIN {X 10.089,Y 331.565,Z -37.417,A 0.015,B 0.000,C 180.000} C_DIS
LIN {X 7.519,Y 325.481,Z -37.661,A 0.015,B 0.000,C 180.000} C_DIS
LIN {X 0.916,Y 325.397,Z -37.905,A 0.015,B -0.000,C 180.000} C_DIS
LIN {X -1.807,Y 331.414,Z -38.149,A 0.015,B 0.000,C 180.000} C_DIS
LIN {X 2.614,Y 336.320,Z -38.393,A 0.015,B 0.000,C -180.000} C_DIS
LIN {X 8.881,Y 334.235,Z -38.637,A 0.015,B 0.000,C -180.000} C_DIS
LIN {X 9.481,Y 327.658,Z -38.881,A 0.015,B 0.000,C -180.000} C_DIS
LIN {X 3.696,Y 324.472,Z -39.125,A 0.015,B 0.000,C -180.000} C_DIS
LIN {X -1.541,Y 328.496,Z -39.369,A 0.015,B 0.000,C 180.000} C_DIS
LIN {X 0.047,Y 334.906,Z -39.613,A 0.015,B 0.000,C -180.000} C_DIS
LIN {X 6.557,Y 336.020,Z -39.857,A 0.015,B -0.000,C 180.000} C_DIS
LIN {X 10.186,Y 330.502,Z -40.101,A 0.015,B 0.000,C -180.000} C_DIS
LIN {X 6.585,Y 324.966,Z -40.345,A 0.015,B 0.000,C -180.000} C_DIS
LIN {X 0.070,Y 326.047,Z -40.589,A 0.015,B 0.000,C 180.000} C_DIS
LIN {X -1.551,Y 332.449,Z -40.833,A 0.015,B 0.000,C -180.000} C_DIS
LIN {X 3.666,Y 336.500,Z -41.077,A 0.015,B 0.000,C 180.000} C_DIS
LIN {X 9.467,Y 333.343,Z -41.321,A 0.015,B 0.000,C 180.000} C_DIS
LIN {X 8.900,Y 326.763,Z -41.565,A 0.015,B 0.000,C -180.000} C_DIS
LIN {X 2.644,Y 324.646,Z -41.810,A 0.015,B 0.000,C -180.000} C_DIS
LIN {X -1.802,Y 329.530,Z -42.054,A 0.015,B -0.000,C -180.000} C_DIS
LIN {X 0.890,Y 335.560,Z -42.298,A 0.015,B -0.000,C -180.000} C_DIS
LIN {X 7.494,Y 335.510,Z -42.542,A 0.015,B -0.000,C -180.000} C_DIS
LIN {X 10.094,Y 329.440,Z -42.786,A 0.015,B 0.000,C 180.000} C_DIS
LIN {X 5.575,Y 324.624,Z -43.030,A 0.015,B 0.000,C -180.000} C_DIS
LIN {X -0.648,Y 326.836,Z -43.274,A 0.015,B -0.000,C 180.000} C_DIS
LIN {X -1.116,Y 333.423,Z -43.518,A 0.015,B 0.000,C 180.000} C_DIS
LIN {X 4.732,Y 336.492,Z -43.762,A 0.015,B 0.000,C -180.000} C_DIS
LIN {X 9.887,Y 332.363,Z -44.006,A 0.015,B 0.000,C -180.000} C_DIS
LIN {X 8.170,Y 325.986,Z -44.250,A 0.015,B -0.000,C 180.000} C_DIS
LIN {X 1.639,Y 325.004,Z -44.494,A 0.015,B 0.000,C -180.000} C_DIS
LIN {X -1.878,Y 330.594,Z -44.738,A 0.015,B 0.000,C -180.000} C_DIS
LIN {X 1.834,Y 336.056,Z -44.982,A 0.015,B 0.000,C 180.000} C_DIS
LIN {X 8.326,Y 334.843,Z -45.226,A 0.015,B -0.000,C 180.000} C_DIS
LIN {X 9.817,Y 328.410,Z -45.470,A 0.015,B 0.000,C 180.000} C_DIS
LIN {X 4.520,Y 324.466,Z -45.714,A 0.015,B 0.000,C -180.000} C_DIS
LIN {X -1.216,Y 327.739,Z -45.958,A 0.015,B 0.000,C -180.000} C_DIS
LIN {X -0.516,Y 334.306,Z -46.202,A 0.015,B 0.000,C 180.000} C_DIS
LIN {X 5.781,Y 336.296,Z -46.446,A 0.015,B 0.000,C -180.000} C_DIS
LIN {X 10.128,Y 331.324,Z -46.690,A 0.015,B 0.000,C 180.000} C_DIS
LIN {X 7.314,Y 325.349,Z -46.935,A 0.015,B 0.000,C 180.000} C_DIS
LIN {X 0.712,Y 325.532,Z -47.179,A 0.015,B 0.000,C 180.000} C_DIS
LIN {X -1.765,Y 331.654,Z -47.423,A 0.015,B 0.000,C 180.000} C_DIS
LIN {X 2.851,Y 336.377,Z -47.667,A 0.015,B 0.000,C -180.000} C_DIS
LIN {X 9.028,Y 334.040,Z -47.911,A 0.015,B 0.000,C -180.000} C_DIS
LIN {X 9.363,Y 327.445,Z -48.155,A 0.015,B 0.000,C -180.000} C_DIS
LIN {X 3.454,Y 324.495,Z -48.399,A 0.015,B -0.000,C 180.000} C_DIS
LIN {X -1.617,Y 328.727,Z -48.643,A 0.015,B 0.000,C -180.000} C_DIS
LIN {X 0.229,Y 335.068,Z -48.887,A 0.015,B 0.000,C 180.000} C_DIS
LIN {X 6.779,Y 335.918,Z -49.131,A 0.015,B 0.000,C 180.000} C_DIS
LIN {X 10.182,Y 330.258,Z -49.375,A 0.015,B 0.000,C 180.000} C_DIS
LIN {X 6.360,Y 324.872,Z -49.619,A 0.015,B 0.000,C -180.000} C_DIS
LIN {X -0.106,Y 326.216,Z -49.863,A 0.015,B -0.000,C 180.000} C_DIS
LIN {X -1.467,Y 332.678,Z -50.107,A 0.015,B -0.000,C -180.000} C_DIS
LIN {X 3.909,Y 336.515,Z -50.351,A 0.015,B 0.000,C -180.000} C_DIS
LIN {X 9.578,Y 333.126,Z -50.595,A 0.015,B 0.000,C 180.000} C_DIS
LIN {X 8.745,Y 326.575,Z -50.839,A 0.015,B 0.000,C 180.000} C_DIS
LIN {X 2.409,Y 324.712,Z -51.083,A 0.015,B 0.000,C 180.000} C_DIS
LIN {X -1.836,Y 329.771,Z -51.327,A 0.015,B 0.000,C 180.000} C_DIS
LIN {X 1.098,Y 335.688,Z -51.571,A 0.015,B 0.000,C 180.000} C_DIS
LIN {X 7.694,Y 335.371,Z -51.815,A 0.015,B 0.000,C 180.000} C_DIS
LIN {X 10.047,Y 329.200,Z -52.060,A 0.015,B 0.000,C 180.000} C_DIS
LIN {X 5.336,Y 324.572,Z -52.304,A 0.015,B 0.000,C 180.000} C_DIS
LIN {X -0.792,Y 327.033,Z -52.548,A 0.015,B 0.000,C -180.000} C_DIS
LIN {X -0.993,Y 333.634,Z -52.792,A 0.015,B 0.000,C -180.000} C_DIS
LIN {X 4.975,Y 336.463,Z -53.036,A 0.015,B 0.000,C -180.000} C_DIS
LIN {X 9.958,Y 332.130,Z -53.280,A 0.015,B -0.000,C 180.000} C_DIS
LIN {X 7.985,Y 325.827,Z -53.524,A 0.015,B -0.000,C 180.000} C_DIS
LIN {X 1.419,Y 325.110,Z -53.768,A 0.015,B 0.000,C 180.000} C_DIS
LIN {X -1.869,Y 330.837,Z -54.012,A 0.015,B 0.000,C 180.000} C_DIS
LIN {X 2.061,Y 336.145,Z -54.256,A 0.015,B 0.000,C -180.000} C_DIS
LIN {X 8.499,Y 334.671,Z -54.500,A 0.015,B -0.000,C 180.000} C_DIS
LIN {X 8.169,Y 335.157,Z -54.500,A 0.015,B 0.000,C -180.000} C_DIS
LIN {X 9.898,Y 336.018,Z -54.500,A 0.015,B -0.000,C 180.000} C_DIS
LIN {X 10.072,Y 335.556,Z -54.500,A 0.015,B 0.000,C -180.000} C_DIS
LIN {X 10.265,Y 334.347,Z -54.500,A 0.015,B 0.000,C -180.000} C_DIS
LIN {X 10.273,Y 32.012,Z -54.500,A 0.015,B 0.000,C 180.000} C_DIS
LIN {X 9.409,Y 35.747,Z -54.500,A 0.015,B 0.000,C -180.000} C_DIS
LIN {X 9.299,Y 36.124,Z -54.500,A 0.015,B -0.000,C 180.000} C_DIS
LIN {X 8.807,Y 37.500,Z -54.500,A 0.015,B 0.000,C -180.000} C_DIS
LIN {X 8.665,Y 37.838,Z -54.500,A 0.015,B 0.000,C 180.000} C_DIS
LIN {X 7.997,Y 39.214,Z -54.500,A 0.015,B 0.000,C -180.000} C_DIS
LIN {X 7.867,Y 39.456,Z -54.500,A 0.015,B 0.000,C -180.000} C_DIS
LIN {X 2.642,Y 48.312,Z -54.500,A 0.015,B 0.000,C -180.000} C_DIS
LIN {X 2.365,Y 48.712,Z -54.500,A 0.015,B 0.000,C 180.000} C_DIS
LIN {X 1.126,Y 50.254,Z -54.500,A 0.015,B 0.000,C -180.000} C_DIS
LIN {X 0.800,Y 50.605,Z -54.500,A 0.015,B -0.000,C 180.000} C_DIS
LIN {X 0.004,Y 51.351,Z -54.500,A 0.015,B 0.000,C 180.000} C_DIS
LIN {X -1.841,Y 53.241,Z -54.500,A 0.015,B 0.000,C 180.000} C_DIS
LIN {X -1.943,Y 53.342,Z -54.500,A 0.015,B 0.000,C -180.000} C_DIS
LIN {X -4.337,Y 55.595,Z -54.500,A 0.015,B 0.000,C 180.000} C_DIS
LIN {X -4.525,Y 55.760,Z -54.500,A 0.015,B 0.000,C -180.000} C_DIS
LIN {X -7.198,Y 57.927,Z -54.500,A 0.015,B 0.000,C -180.000} C_DIS
LIN {X -7.354,Y 58.046,Z -54.500,A 0.015,B -0.000,C 180.000} C_DIS
LIN {X -117.499,Y 137.197,Z -54.500,A 0.015,B 0.000,C 180.000} C_DIS
LIN {X -117.959,Y 137.475,Z -54.500,A 0.015,B 0.000,C -180.000} C_DIS
LIN {X -119.420,Y 138.206,Z -54.500,A 0.015,B 0.000,C 180.000} C_DIS
LIN {X -120.056,Y 138.448,Z -54.500,A 0.015,B 0.000,C -180.000} C_DIS
LIN {X -121.507,Y 138.838,Z -54.500,A 0.015,B 0.000,C -180.000} C_DIS
LIN {X -122.106,Y 138.942,Z -54.500,A 0.015,B 0.000,C -180.000} C_DIS
LIN {X -123.558,Y 139.062,Z -54.500,A 0.015,B -0.000,C -180.000} C_DIS
LIN {X -124.202,Y 139.053,Z -54.500,A 0.015,B 0.000,C -180.000} C_DIS
LIN {X -126.741,Y 138.777,Z -54.500,A 0.015,B 0.000,C 180.000} C_DIS
LIN {X -127.229,Y 138.687,Z -54.500,A 0.015,B -0.000,C -180.000} C_DIS
LIN {X -129.405,Y 138.119,Z -54.500,A 0.015,B 0.000,C -180.000} C_DIS
LIN {X -129.666,Y 138.040,Z -54.500,A 0.015,B 0.000,C 180.000} C_DIS
LIN {X -131.117,Y 137.534,Z -54.500,A 0.015,B -0.000,C 180.000} C_DIS
LIN {X -131.374,Y 137.432,Z -54.500,A 0.015,B 0.000,C 180.000} C_DIS
LIN {X -134.374,Y 136.102,Z -54.500,A 0.015,B 0.000,C 180.000} C_DIS
LIN {X -134.690,Y 135.941,Z -54.500,A 0.015,B 0.000,C -180.000} C_DIS
LIN {X -171.123,Y 114.978,Z -54.500,A 0.015,B 0.000,C 180.000} C_DIS
LIN {X -171.775,Y 114.489,Z -54.500,A 0.015,B 0.000,C 180.000} C_DIS
LIN {X -172.532,Y 113.765,Z -54.500,A 0.015,B 0.000,C -180.000} C_DIS
CIRC {X -172.869,Y 113.390,Z -54.500,A 0.015,B 0.000,C -180.000},{X -173.146,Y 112.970,Z -54.500,A 0.015,B -0.000,C 180.000} C_DIS
LIN {X -173.640,Y 112.084,Z -54.500,A 0.015,B -0.000,C 180.000} C_DIS
CIRC {X -173.858,Y 111.612,Z -54.500,A 0.015,B 0.000,C 180.000},{X -174.000,Y 111.113,Z -54.500,A 0.015,B 0.000,C -180.000} C_DIS
LIN {X -174.222,Y 110.024,Z -54.500,A 0.015,B 0.000,C 180.000} C_DIS
CIRC {X -174.287,Y 109.489,Z -54.500,A 0.015,B -0.000,C 180.000},{X -174.267,Y 108.949,Z -54.500,A 0.015,B 0.000,C -180.000} C_DIS
LIN {X -174.137,Y 107.861,Z -54.500,A 0.015,B 0.000,C -180.000} C_DIS
CIRC {X -174.027,Y 107.317,Z -54.500,A 0.015,B 0.000,C -180.000},{X -173.829,Y 106.799,Z -54.500,A 0.015,B 0.000,C -180.000} C_DIS
LIN {X -173.323,Y 105.742,Z -54.500,A 0.015,B 0.000,C -180.000} C_DIS
CIRC {X -173.058,Y 105.286,Z -54.500,A 0.015,B 0.000,C -180.000},{X -172.726,Y 104.876,Z -54.500,A 0.015,B 0.000,C 180.000} C_DIS
LIN {X -172.049,Y 104.161,Z -54.500,A 0.015,B 0.000,C 180.000} C_DIS
LIN {X -171.285,Y 103.559,Z -54.500,A 0.015,B 0.000,C -180.000} C_DIS
LIN {X -55.841,Y 36.985,Z -54.500,A 0.015,B 0.000,C 180.000} C_DIS
LIN {X -63.759,Y 23.290,Z -54.500,A 0.015,B 0.000,C 180.000} C_DIS
LIN {X -178.737,Y 89.791,Z -54.500,A 0.015,B -0.000,C -180.000} C_DIS
LIN {X -179.265,Y 90.038,Z -54.500,A 0.015,B 0.000,C 180.000} C_DIS
LIN {X -180.241,Y 90.396,Z -54.500,A 0.015,B 0.000,C -180.000} C_DIS
CIRC {X -180.730,Y 90.535,Z -54.500,A 0.015,B 0.000,C 180.000},{X -181.235,Y 90.599,Z -54.500,A 0.015,B 0.000,C 180.000} C_DIS
LIN {X -182.275,Y 90.651,Z -54.500,A 0.015,B 0.000,C -180.000} C_DIS
CIRC {X -182.788,Y 90.638,Z -54.500,A 0.015,B 0.000,C 180.000},{X -183.294,Y 90.548,Z -54.500,A 0.015,B -0.000,C -180.000} C_DIS
LIN {X -184.317,Y 90.283,Z -54.500,A 0.015,B -0.000,C -180.000} C_DIS
CIRC {X -184.812,Y 90.113,Z -54.500,A 0.015,B 0.000,C 180.000},{X -185.274,Y 89.870,Z -54.500,A 0.015,B 0.000,C -180.000} C_DIS
LIN {X -186.187,Y 89.294,Z -54.500,A 0.015,B -0.000,C 180.000} C_DIS
LIN {X -186.718,Y 88.880,Z -54.500,A 0.015,B 0.000,C 180.000} C_DIS
LIN {X -186.934,Y 88.674,Z -54.500,A 0.015,B 0.000,C 180.000} C_DIS
LIN {X -187.388,Y 88.140,Z -54.500,A 0.015,B -0.000,C 180.000} C_DIS
LIN {X -188.033,Y 87.200,Z -54.500,A 0.015,B 0.000,C 180.000} C_DIS
CIRC {X -188.295,Y 86.744,Z -54.500,A 0.015,B -0.000,C 180.000},{X -188.484,Y 86.254,Z -54.500,A 0.015,B 0.000,C -180.000} C_DIS
LIN {X -188.773,Y 85.285,Z -54.500,A 0.015,B 0.000,C -180.000} C_DIS
LIN {X -188.914,Y 84.317,Z -54.500,A 0.015,B 0.000,C 180.000} C_DIS
LIN {X -188.884,Y 42.238,Z -54.500,A 0.015,B 0.000,C 180.000} C_DIS
LIN {X -188.867,Y 41.908,Z -54.500,A 0.015,B 0.000,C -180.000} C_DIS
LIN {X -188.581,Y 39.006,Z -54.500,A 0.015,B -0.000,C 180.000} C_DIS
LIN {X -188.535,Y 38.692,Z -54.500,A 0.015,B -0.000,C 180.000} C_DIS
LIN {X -187.970,Y 35.790,Z -54.500,A 0.015,B 0.000,C 180.000} C_DIS
LIN {X -187.880,Y 35.431,Z -54.500,A 0.015,B 0.000,C 180.000} C_DIS
LIN {X -187.428,Y 33.980,Z -54.500,A 0.015,B 0.000,C 180.000} C_DIS
LIN {X -187.306,Y 33.649,Z -54.500,A 0.015,B 0.000,C -180.000} C_DIS
LIN {X -186.621,Y 32.056,Z -54.500,A 0.015,B 0.000,C 180.000} C_DIS
LIN {X -186.433,Y 31.684,Z -54.500,A 0.015,B 0.000,C 180.000} C_DIS
LIN {X -185.667,Y 30.375,Z -54.500,A 0.015,B 0.000,C -180.000} C_DIS
LIN {X -185.335,Y 29.905,Z -54.500,A 0.015,B -0.000,C 180.000} C_DIS
LIN {X -184.358,Y 28.744,Z -54.500,A 0.015,B -0.000,C 180.000} C_DIS
LIN {X -183.776,Y 28.199,Z -54.500,A 0.015,B -0.000,C 180.000} C_DIS
LIN {X -182.333,Y 27.136,Z -54.500,A 0.015,B 0.000,C 180.000} C_DIS
LIN {X -181.720,Y 26.777,Z -54.500,A 0.015,B -0.000,C 180.000} C_DIS
LIN {X -60.289,Y -28.089,Z -54.500,A 0.015,B 0.000,C 180.000} C_DIS
LIN {X -60.240,Y -28.111,Z -54.500,A 0.015,B 0.000,C 180.000} C_DIS
LIN {X -55.886,Y -29.995,Z -54.500,A 0.015,B -0.000,C 180.000} C_DIS
LIN {X -55.590,Y -30.107,Z -54.500,A 0.015,B 0.000,C 180.000} C_DIS
LIN {X -52.030,Y -31.266,Z -54.500,A 0.015,B 0.000,C -180.000} C_DIS
LIN {X -341.507,Y -31.266,Z -54.500,A 0.015,B 0.000,C -180.000} C_DIS
LIN {X -339.421,Y -30.621,Z -54.500,A 0.015,B 0.000,C 180.000} C_DIS
LIN {X -339.236,Y -30.558,Z -54.500,A 0.015,B 0.000,C -180.000} C_DIS
LIN {X -336.334,Y -29.473,Z -54.500,A 0.015,B -0.000,C -180.000} C_DIS
LIN {X -336.126,Y -29.388,Z -54.500,A 0.015,B 0.000,C -180.000} C_DIS
LIN {X -212.259,Y 26.520,Z -54.500,A 0.015,B 0.000,C 180.000} C_DIS
LIN {X -211.788,Y 26.780,Z -54.500,A 0.015,B -0.000,C 180.000} C_DIS
LIN {X -210.122,Y 27.879,Z -54.500,A 0.015,B 0.000,C 180.000} C_DIS
LIN {X -209.548,Y 28.357,Z -54.500,A 0.015,B -0.000,C -180.000} C_DIS
LIN {X -208.778,Y 29.158,Z -54.500,A 0.015,B 0.000,C 180.000} C_DIS
LIN {X -208.443,Y 29.566,Z -54.500,A 0.015,B 0.000,C 180.000} C_DIS
LIN {X -207.434,Y 31.010,Z -54.500,A 0.015,B 0.000,C 180.000} C_DIS
LIN {X -207.108,Y 31.590,Z -54.500,A 0.015,B 0.000,C 180.000} C_DIS
LIN {X -206.215,Y 33.628,Z -54.500,A 0.015,B -0.000,C 180.000} C_DIS
LIN {X -206.084,Y 33.980,Z -54.500,A 0.015,B -0.000,C 180.000} C_DIS
LIN {X -205.632,Y 35.431,Z -54.500,A 0.015,B -0.000,C 180.000} C_DIS
LIN {X -205.542,Y 35.790,Z -54.500,A 0.015,B -0.000,C 180.000} C_DIS
LIN {X -204.977,Y 38.692,Z -54.500,A 0.015,B 0.000,C -180.000} C_DIS
LIN {X -204.931,Y 39.006,Z -54.500,A 0.015,B 0.000,C -180.000} C_DIS
LIN {X -204.645,Y 41.908,Z -54.500,A 0.015,B 0.000,C -180.000} C_DIS
LIN {X -204.628,Y 42.238,Z -54.500,A 0.015,B 0.000,C -180.000} C_DIS
LIN {X -204.598,Y 84.317,Z -54.500,A 0.015,B 0.000,C 180.000} C_DIS
LIN {X -204.739,Y 85.285,Z -54.500,A 0.015,B -0.000,C 180.000} C_DIS
LIN {X -205.028,Y 86.254,Z -54.500,A 0.015,B 0.000,C 180.000} C_DIS
CIRC {X -205.217,Y 86.744,Z -54.500,A 0.015,B 0.000,C 180.000},{X -205.479,Y 87.200,Z -54.500,A 0.015,B 0.000,C -180.000} C_DIS
LIN {X -206.123,Y 88.140,Z -54.500,A 0.015,B -0.000,C -180.000} C_DIS
CIRC {X -206.473,Y 88.570,Z -54.500,A 0.015,B 0.000,C -180.000},{X -206.889,Y 88.937,Z -54.500,A 0.015,B -0.000,C 180.000} C_DIS
LIN {X -207.792,Y 89.612,Z -54.500,A 0.015,B 0.000,C 180.000} C_DIS
CIRC {X -208.223,Y 89.885,Z -54.500,A 0.015,B 0.000,C -180.000},{X -208.689,Y 90.091,Z -54.500,A 0.015,B 0.000,C 180.000} C_DIS
LIN {X -209.592,Y 90.410,Z -54.500,A 0.015,B 0.000,C -180.000} C_DIS
LIN {X -210.548,Y 90.599,Z -54.500,A 0.015,B -0.000,C 180.000} C_DIS
LIN {X -211.588,Y 90.651,Z -54.500,A 0.015,B 0.000,C -180.000} C_DIS
LIN {X -212.574,Y 90.556,Z -54.500,A 0.015,B -0.000,C 180.000} C_DIS
LIN {X -213.533,Y 90.318,Z -54.500,A 0.015,B 0.000,C -180.000} C_DIS
LIN {X -214.411,Y 89.964,Z -54.500,A 0.015,B 0.000,C 180.000} C_DIS
LIN {X -329.752,Y 23.290,Z -54.500,A 0.015,B 0.000,C 180.000} C_DIS
LIN {X -337.671,Y 36.985,Z -54.500,A 0.015,B 0.000,C 180.000} C_DIS
LIN {X -222.227,Y 103.559,Z -54.500,A 0.015,B 0.000,C 180.000} C_DIS
LIN {X -221.463,Y 104.161,Z -54.500,A 0.015,B 0.000,C -180.000} C_DIS
LIN {X -220.786,Y 104.876,Z -54.500,A 0.015,B 0.000,C 180.000} C_DIS
CIRC {X -220.453,Y 105.286,Z -54.500,A 0.015,B -0.000,C 180.000},{X -220.189,Y 105.742,Z -54.500,A 0.015,B -0.000,C -180.000} C_DIS
LIN {X -219.683,Y 106.799,Z -54.500,A 0.015,B 0.000,C -180.000} C_DIS
CIRC {X -219.485,Y 107.317,Z -54.500,A 0.015,B 0.000,C -180.000},{X -219.375,Y 107.861,Z -54.500,A 0.015,B 0.000,C -180.000} C_DIS
LIN {X -219.245,Y 108.949,Z -54.500,A 0.015,B -0.000,C -180.000} C_DIS
CIRC {X -219.224,Y 109.489,Z -54.500,A 0.015,B 0.000,C 180.000},{X -219.290,Y 110.024,Z -54.500,A 0.015,B 0.000,C 180.000} C_DIS
LIN {X -219.512,Y 111.113,Z -54.500,A 0.015,B 0.000,C -180.000} C_DIS
CIRC {X -219.654,Y 111.612,Z -54.500,A 0.015,B -0.000,C 180.000},{X -219.872,Y 112.084,Z -54.500,A 0.015,B 0.000,C 180.000} C_DIS
LIN {X -220.366,Y 112.970,Z -54.500,A 0.015,B 0.000,C -180.000} C_DIS
CIRC {X -220.643,Y 113.390,Z -54.500,A 0.015,B 0.000,C 180.000},{X -220.980,Y 113.765,Z -54.500,A 0.015,B 0.000,C -180.000} C_DIS
LIN {X -221.736,Y 114.489,Z -54.500,A 0.015,B 0.000,C -180.000} C_DIS
LIN {X -222.389,Y 114.978,Z -54.500,A 0.015,B 0.000,C 180.000} C_DIS
LIN {X -258.145,Y 135.553,Z -54.500,A 0.015,B -0.000,C 180.000} C_DIS
LIN {X -258.301,Y 135.637,Z -54.500,A 0.015,B 0.000,C -180.000} C_DIS
LIN {X -260.330,Y 136.668,Z -54.500,A 0.015,B 0.000,C -180.000} C_DIS
LIN {X -260.646,Y 136.809,Z -54.500,A 0.015,B 0.000,C -180.000} C_DIS
LIN {X -263.744,Y 138.002,Z -54.500,A 0.015,B 0.000,C 180.000} C_DIS
LIN {X -264.106,Y 138.119,Z -54.500,A 0.015,B 0.000,C -180.000} C_DIS
LIN {X -266.283,Y 138.687,Z -54.500,A 0.015,B 0.000,C 180.000} C_DIS
LIN {X -266.726,Y 138.772,Z -54.500,A 0.015,B -0.000,C -180.000} C_DIS
LIN {X -268.903,Y 139.038,Z -54.500,A 0.015,B 0.000,C 180.000} C_DIS
LIN {X -269.443,Y 139.060,Z -54.500,A 0.015,B -0.000,C 180.000} C_DIS
LIN {X -270.894,Y 139.005,Z -54.500,A 0.015,B 0.000,C -180.000} C_DIS
LIN {X -271.453,Y 138.937,Z -54.500,A 0.015,B 0.000,C -180.000} C_DIS
LIN {X -272.904,Y 138.635,Z -54.500,A 0.015,B 0.000,C -180.000} C_DIS
LIN {X -273.608,Y 138.406,Z -54.500,A 0.015,B 0.000,C -180.000} C_DIS
LIN {X -275.059,Y 137.751,Z -54.500,A 0.015,B 0.000,C 180.000} C_DIS
LIN {X -275.640,Y 137.416,Z -54.500,A 0.015,B 0.000,C -180.000} C_DIS
LIN {X -382.147,Y 60.929,Z -54.500,A 0.015,B 0.000,C -180.000} C_DIS
LIN {X -387.521,Y 56.988,Z -54.500,A 0.015,B 0.000,C 180.000} C_DIS
LIN {X -387.767,Y 56.789,Z -54.500,A 0.015,B 0.000,C 180.000} C_DIS
LIN {X -390.954,Y 53.958,Z -54.500,A 0.015,B 0.000,C 180.000} C_DIS
LIN {X -391.168,Y 53.750,Z -54.500,A 0.015,B 0.000,C 180.000} C_DIS
LIN {X -392.888,Y 51.928,Z -54.500,A 0.015,B 0.000,C -180.000} C_DIS
LIN {X -394.004,Y 50.941,Z -54.500,A 0.015,B -0.000,C -180.000} C_DIS
LIN {X -394.386,Y 50.543,Z -54.500,A 0.015,B 0.000,C 180.000} C_DIS
LIN {X -395.864,Y 48.729,Z -54.500,A 0.015,B 0.000,C -180.000} C_DIS
LIN {X -396.111,Y 48.383,Z -54.500,A 0.015,B -0.000,C -180.000} C_DIS
LIN {X -397.016,Y 46.932,Z -54.500,A 0.015,B -0.000,C 180.000} C_DIS
LIN {X -397.070,Y 46.842,Z -54.500,A 0.015,B -0.000,C 180.000} C_DIS
LIN {X -401.776,Y 38.750,Z -54.500,A 0.015,B 0.000,C 180.000} C_DIS
LIN {X -401.996,Y 38.296,Z -54.500,A 0.015,B -0.000,C -180.000} C_DIS
LIN {X -402.678,Y 36.576,Z -54.500,A 0.015,B 0.000,C -180.000} C_DIS
LIN {X -402.827,Y 36.100,Z -54.500,A 0.015,B -0.000,C 180.000} C_DIS
LIN {X -403.779,Y 32.037,Z -54.500,A 0.015,B 0.000,C 180.000} C_DIS
LIN {X -403.787,Y 333.800,Z -54.500,A 0.015,B -0.000,C -180.000} C_DIS
LIN {X -403.730,Y 334.871,Z -54.500,A 0.015,B 0.000,C 180.000} C_DIS
LIN {X -403.533,Y 335.736,Z -54.500,A 0.015,B 0.000,C 180.000} C_DIS
LIN {X -403.418,Y 336.003,Z -54.500,A 0.015,B 0.000,C -180.000} C_DIS
LIN {X -403.212,Y 336.308,Z -54.500,A 0.015,B 0.000,C 180.000} C_DIS
LIN {X -400.955,Y 338.598,Z -54.500,A 0.015,B 0.000,C -180.000} C_DIS
LIN {X -400.596,Y 338.832,Z -54.500,A 0.015,B 0.000,C 180.000} C_DIS
LIN {X -400.134,Y 339.006,Z -54.500,A 0.015,B 0.000,C 180.000} C_DIS
LIN {X -398.924,Y 339.199,Z -54.500,A 0.015,B -0.000,C -180.000} C_DIS
LIN {X -213.439,Y 339.203,Z -54.500,A 0.015,B 0.000,C -180.000} C_DIS
LIN {X -213.596,Y 339.165,Z -54.500,A 0.015,B -0.000,C -180.000} C_DIS
LIN {X -214.684,Y 338.873,Z -54.500,A 0.015,B -0.000,C 180.000} C_DIS
LIN {X -215.273,Y 338.655,Z -54.500,A 0.015,B -0.000,C -180.000} C_DIS
LIN {X -225.794,Y 333.594,Z -54.500,A 0.015,B 0.000,C -180.000} C_DIS
LIN {X -226.167,Y 333.385,Z -54.500,A 0.015,B -0.000,C 180.000} C_DIS
LIN {X -227.618,Y 332.445,Z -54.500,A 0.015,B 0.000,C 180.000} C_DIS
LIN {X -228.088,Y 332.078,Z -54.500,A 0.015,B 0.000,C -180.000} C_DIS
LIN {X -236.316,Y 324.390,Z -54.500,A 0.015,B 0.000,C 180.000} C_DIS
LIN {X -236.659,Y 324.018,Z -54.500,A 0.015,B 0.000,C 180.000} C_DIS
LIN {X -238.095,Y 322.204,Z -54.500,A 0.015,B 0.000,C -180.000} C_DIS
LIN {X -238.387,Y 321.769,Z -54.500,A 0.015,B 0.000,C 180.000} C_DIS
LIN {X -243.718,Y 312.338,Z -54.500,A 0.015,B 0.000,C -180.000} C_DIS
LIN {X -243.927,Y 311.897,Z -54.500,A 0.015,B 0.000,C 180.000} C_DIS
LIN {X -244.631,Y 310.083,Z -54.500,A 0.015,B 0.000,C -180.000} C_DIS
LIN {X -244.781,Y 309.583,Z -54.500,A 0.015,B 0.000,C -180.000} C_DIS
LIN {X -245.073,Y 308.251,Z -54.500,A 0.015,B 0.000,C -180.000} C_DIS
LIN {X -245.794,Y 305.837,Z -54.500,A 0.015,B 0.000,C -180.000} C_DIS
LIN {X -245.851,Y 305.619,Z -54.500,A 0.015,B 0.000,C -180.000} C_DIS
LIN {X -246.510,Y 302.717,Z -54.500,A 0.015,B 0.000,C 180.000} C_DIS
LIN {X -246.546,Y 302.535,Z -54.500,A 0.015,B 0.000,C 180.000} C_DIS
LIN {X -247.040,Y 299.633,Z -54.500,A 0.015,B 0.000,C 180.000} C_DIS
LIN {X -247.071,Y 299.402,Z -54.500,A 0.015,B -0.000,C -180.000} C_DIS
LIN {X -260.627,Y 163.734,Z -54.500,A 0.015,B -0.000,C 180.000} C_DIS
LIN {X -260.634,Y 163.131,Z -54.500,A 0.015,B -0.000,C 180.000} C_DIS
LIN {X -260.490,Y 161.317,Z -54.500,A 0.015,B 0.000,C -180.000} C_DIS
LIN {X -260.358,Y 160.615,Z -54.500,A 0.015,B 0.000,C 180.000} C_DIS
LIN {X -260.033,Y 159.526,Z -54.500,A 0.015,B 0.000,C -180.000} C_DIS
LIN {X -259.867,Y 159.087,Z -54.500,A 0.015,B -0.000,C -180.000} C_DIS
LIN {X -259.328,Y 157.910,Z -54.500,A 0.015,B 0.000,C 180.000} C_DIS
LIN {X -259.028,Y 157.385,Z -54.500,A 0.015,B -0.000,C -180.000} C_DIS
LIN {X -257.747,Y 155.547,Z -54.500,A 0.015,B 0.000,C 180.000} C_DIS
LIN {X -257.463,Y 155.193,Z -54.500,A 0.015,B 0.000,C 180.000} C_DIS
LIN {X -255.842,Y 153.428,Z -54.500,A 0.015,B 0.000,C -180.000} C_DIS
LIN {X -255.531,Y 153.131,Z -54.500,A 0.015,B 0.000,C -180.000} C_DIS
LIN {X -253.455,Y 151.381,Z -54.500,A 0.015,B 0.000,C -180.000} C_DIS
LIN {X -253.223,Y 151.202,Z -54.500,A 0.015,B 0.000,C 180.000} C_DIS
LIN {X -250.945,Y 149.597,Z -54.500,A 0.015,B -0.000,C -180.000} C_DIS
LIN {X -250.691,Y 149.434,Z -54.500,A 0.015,B 0.000,C 180.000} C_DIS
LIN {X -214.412,Y 128.454,Z -54.500,A 0.015,B 0.000,C 180.000} C_DIS
CIRC {X -213.956,Y 128.234,Z -54.500,A 0.015,B -0.000,C 180.000},{X -213.472,Y 128.085,Z -54.500,A 0.015,B -0.000,C 180.000} C_DIS
LIN {X -212.383,Y 127.836,Z -54.500,A 0.015,B 0.000,C 180.000} C_DIS
CIRC {X -211.849,Y 127.758,Z -54.500,A 0.015,B 0.000,C 180.000},{X -211.308,Y 127.766,Z -54.500,A 0.015,B 0.000,C 180.000} C_DIS
LIN {X -210.220,Y 127.871,Z -54.500,A 0.015,B -0.000,C -180.000} C_DIS
CIRC {X -209.684,Y 127.966,Z -54.500,A 0.015,B 0.000,C 180.000},{X -209.171,Y 128.146,Z -54.500,A 0.015,B 0.000,C 180.000} C_DIS
LIN {X -208.138,Y 128.604,Z -54.500,A 0.015,B 0.000,C 180.000} C_DIS
LIN {X -207.316,Y 129.120,Z -54.500,A 0.015,B -0.000,C -180.000} C_DIS
LIN {X -206.661,Y 129.678,Z -54.500,A 0.015,B 0.000,C 180.000} C_DIS
LIN {X -206.044,Y 130.371,Z -54.500,A 0.015,B 0.000,C 180.000} C_DIS
LIN {X -205.464,Y 131.236,Z -54.500,A 0.015,B -0.000,C -180.000} C_DIS
LIN {X -205.047,Y 132.107,Z -54.500,A 0.015,B -0.000,C -180.000} C_DIS
LIN {X -204.766,Y 133.004,Z -54.500,A 0.015,B 0.000,C 180.000} C_DIS
CIRC {X -204.650,Y 133.505,Z -54.500,A 0.015,B 0.000,C 180.000},{X -204.611,Y 134.017,Z -54.500,A 0.015,B 0.000,C 180.000} C_DIS
LIN {X -204.666,Y 267.359,Z -54.500,A 0.015,B 0.000,C 180.000} C_DIS
LIN {X -188.846,Y 267.359,Z -54.500,A 0.015,B 0.000,C 180.000} C_DIS
LIN {X -188.901,Y 134.017,Z -54.500,A 0.015,B -0.000,C -180.000} C_DIS
CIRC {X -188.862,Y 133.505,Z -54.500,A 0.015,B 0.000,C 180.000},{X -188.746,Y 133.004,Z -54.500,A 0.015,B 0.000,C 180.000} C_DIS
LIN {X -188.465,Y 132.107,Z -54.500,A 0.015,B 0.000,C -180.000} C_DIS
LIN {X -188.047,Y 131.236,Z -54.500,A 0.015,B -0.000,C 180.000} C_DIS
LIN {X -187.468,Y 130.371,Z -54.500,A 0.015,B -0.000,C -180.000} C_DIS
LIN {X -186.851,Y 129.678,Z -54.500,A 0.015,B 0.000,C -180.000} C_DIS
LIN {X -186.196,Y 129.120,Z -54.500,A 0.015,B 0.000,C -180.000} C_DIS
LIN {X -185.374,Y 128.604,Z -54.500,A 0.015,B 0.000,C 180.000} C_DIS
LIN {X -184.341,Y 128.146,Z -54.500,A 0.015,B 0.000,C -180.000} C_DIS
CIRC {X -183.828,Y 127.966,Z -54.500,A 0.015,B 0.000,C 180.000},{X -183.292,Y 127.871,Z -54.500,A 0.015,B -0.000,C 180.000} C_DIS
LIN {X -182.204,Y 127.766,Z -54.500,A 0.015,B 0.000,C 180.000} C_DIS
CIRC {X -181.663,Y 127.758,Z -54.500,A 0.015,B -0.000,C -180.000},{X -181.129,Y 127.836,Z -54.500,A 0.015,B 0.000,C -180.000} C_DIS
LIN {X -180.040,Y 128.085,Z -54.500,A 0.015,B 0.000,C 180.000} C_DIS
CIRC {X -179.556,Y 128.234,Z -54.500,A 0.015,B 0.000,C 180.000},{X -179.100,Y 128.454,Z -54.500,A 0.015,B 0.000,C -180.000} C_DIS
LIN {X -142.821,Y 149.434,Z -54.500,A 0.015,B -0.000,C -180.000} C_DIS
LIN {X -142.611,Y 149.566,Z -54.500,A 0.015,B 0.000,C -180.000} C_DIS
LIN {X -141.160,Y 150.554,Z -54.500,A 0.015,B 0.000,C 180.000} C_DIS
LIN {X -140.926,Y 150.729,Z -54.500,A 0.015,B -0.000,C -180.000} C_DIS
LIN {X -138.024,Y 153.095,Z -54.500,A 0.015,B -0.000,C 180.000} C_DIS
LIN {X -137.731,Y 153.364,Z -54.500,A 0.015,B 0.000,C 180.000} C_DIS
LIN {X -136.616,Y 154.516,Z -54.500,A 0.015,B 0.000,C 180.000} C_DIS
LIN {X -136.369,Y 154.801,Z -54.500,A 0.015,B 0.000,C -180.000} C_DIS
LIN {X -134.949,Y 156.639,Z -54.500,A 0.015,B -0.000,C 180.000} C_DIS
LIN {X -134.648,Y 157.102,Z -54.500,A 0.015,B 0.000,C -180.000} C_DIS
LIN {X -133.879,Y 158.529,Z -54.500,A 0.015,B 0.000,C -180.000} C_DIS
LIN {X -133.634,Y 159.105,Z -54.500,A 0.015,B 0.000,C 180.000} C_DIS
LIN {X -133.171,Y 160.556,Z -54.500,A 0.015,B 0.000,C 180.000} C_DIS
LIN {X -133.022,Y 161.317,Z -54.500,A 0.015,B -0.000,C -180.000} C_DIS
LIN {X -132.878,Y 163.131,Z -54.500,A 0.015,B 0.000,C 180.000} C_DIS
LIN {X -132.885,Y 163.734,Z -54.500,A 0.015,B 0.000,C 180.000} C_DIS
LIN {X -145.505,Y 290.232,Z -54.500,A 0.015,B -0.000,C -180.000} C_DIS
LIN {X -146.648,Y 300.877,Z -54.500,A 0.015,B 0.000,C 180.000} C_DIS
LIN {X -146.703,Y 301.224,Z -54.500,A 0.015,B -0.000,C 180.000} C_DIS
LIN {X -147.479,Y 304.852,Z -54.500,A 0.015,B 0.000,C -180.000} C_DIS
LIN {X -147.539,Y 305.090,Z -54.500,A 0.015,B -0.000,C 180.000} C_DIS
LIN {X -148.333,Y 307.816,Z -54.500,A 0.015,B 0.000,C 180.000} C_DIS
LIN {X -148.497,Y 308.731,Z -54.500,A 0.015,B 0.000,C -180.000} C_DIS
LIN {X -148.643,Y 309.278,Z -54.500,A 0.015,B -0.000,C 180.000} C_DIS
LIN {X -149.555,Y 311.817,Z -54.500,A 0.015,B -0.000,C -180.000} C_DIS
LIN {X -149.794,Y 312.338,Z -54.500,A 0.015,B 0.000,C -180.000} C_DIS
LIN {X -155.125,Y 321.769,Z -54.500,A 0.015,B -0.000,C 180.000} C_DIS
LIN {X -155.417,Y 322.204,Z -54.500,A 0.015,B 0.000,C 180.000} C_DIS
LIN {X -156.853,Y 324.018,Z -54.500,A 0.015,B 0.000,C 180.000} C_DIS
LIN {X -157.193,Y 324.387,Z -54.500,A 0.015,B 0.000,C -180.000} C_DIS
LIN {X -165.058,Y 331.756,Z -54.500,A 0.015,B 0.000,C 180.000} C_DIS
LIN {X -165.368,Y 332.013,Z -54.500,A 0.015,B 0.000,C -180.000} C_DIS
LIN {X -166.819,Y 333.079,Z -54.500,A 0.015,B 0.000,C 180.000} C_DIS
LIN {X -167.345,Y 333.397,Z -54.500,A 0.015,B -0.000,C -180.000} C_DIS
LIN {X -177.866,Y 338.501,Z -54.500,A 0.015,B -0.000,C -180.000} C_DIS
LIN {X -178.252,Y 338.659,Z -54.500,A 0.015,B 0.000,C -180.000} C_DIS
LIN {X -179.341,Y 339.030,Z -54.500,A 0.015,B 0.000,C 180.000} C_DIS
LIN {X -179.926,Y 339.172,Z -54.500,A 0.015,B -0.000,C -180.000} C_DIS
LIN {X -180.137,Y 339.204,Z -54.500,A 0.015,B 0.000,C -180.000} C_DIS
LIN {X 4.865,Y 339.209,Z -54.500,A 0.015,B 0.000,C -180.000} C_DIS
LIN {X 5.937,Y 339.152,Z -54.500,A 0.015,B -0.000,C -180.000} C_DIS
LIN {X 6.802,Y 338.955,Z -54.500,A 0.015,B 0.000,C -180.000} C_DIS
LIN {X 7.069,Y 338.840,Z -54.500,A 0.015,B -0.000,C -180.000} C_DIS
LIN {X 7.566,Y 338.456,Z -54.330,A 0.015,B 0.000,C 180.000} C_DIS
LIN {X 7.779,Y 338.046,Z -53.865,A 0.015,B -0.000,C 180.000} C_DIS
LIN {X 7.818,Y 337.880,Z -53.230,A 0.015,B 0.000,C -180.000} C_DIS
$VEL.CP = 1.00000
LIN {X 7.818,Y 337.880,Z 11.000,A 0.015,B -0.000,C 180.000} C_DIS
$VEL.CP = 1.00000
LIN {X -66.822,Y 254.064,Z 11.000,A 0.015,B 0.000,C -180.000} C_DIS
$VEL.CP = 1.00000
LIN {X -66.822,Y 254.064,Z -42.731,A 0.015,B 0.000,C 180.000} C_DIS
$VEL.CP = 0.10000
LIN {X -66.660,Y 254.045,Z -43.353,A 0.015,B 0.000,C 180.000} C_DIS
LIN {X -66.214,Y 254.017,Z -43.816,A 0.015,B -0.000,C -180.000} C_DIS
LIN {X -65.599,Y 254.032,Z -44.000,A 0.015,B 0.000,C -180.000} C_DIS
LIN {X -60.362,Y 258.056,Z -44.244,A 0.015,B 0.000,C -180.000} C_DIS
LIN {X -61.951,Y 264.467,Z -44.488,A 0.015,B 0.000,C -180.000} C_DIS
LIN {X -68.460,Y 265.580,Z -44.732,A 0.015,B -0.000,C 180.000} C_DIS
LIN {X -72.089,Y 260.062,Z -44.976,A 0.015,B 0.000,C -180.000} C_DIS
LIN {X -68.487,Y 254.526,Z -45.220,A 0.015,B 0.000,C 180.000} C_DIS
LIN {X -61.972,Y 255.608,Z -45.464,A 0.015,B 0.000,C 180.000} C_DIS
LIN {X -60.352,Y 262.010,Z -45.708,A 0.015,B 0.000,C -180.000} C_DIS
LIN {X -65.569,Y 266.060,Z -45.952,A 0.015,B 0.000,C 180.000} C_DIS
LIN {X -71.370,Y 262.903,Z -46.196,A 0.015,B 0.000,C 180.000} C_DIS
LIN {X -70.802,Y 256.323,Z -46.440,A 0.015,B 0.000,C 180.000} C_DIS
LIN {X -64.546,Y 254.207,Z -46.685,A 0.015,B 0.000,C 180.000} C_DIS
LIN {X -60.100,Y 259.091,Z -46.929,A 0.015,B 0.000,C -180.000} C_DIS
LIN {X -62.793,Y 265.121,Z -47.173,A 0.015,B 0.000,C -180.000} C_DIS
LIN {X -69.397,Y 265.070,Z -47.417,A 0.015,B 0.000,C 180.000} C_DIS
LIN {X -71.997,Y 258.999,Z -47.661,A 0.015,B 0.000,C 180.000} C_DIS
LIN {X -67.477,Y 254.184,Z -47.905,A 0.015,B 0.000,C 180.000} C_DIS
LIN {X -61.254,Y 256.397,Z -48.149,A 0.015,B 0.000,C -180.000} C_DIS
LIN {X -60.787,Y 262.984,Z -48.393,A 0.015,B 0.000,C 180.000} C_DIS
LIN {X -66.636,Y 266.052,Z -48.637,A 0.015,B 0.000,C -180.000} C_DIS
LIN {X -71.790,Y 261.923,Z -48.881,A 0.015,B 0.000,C -180.000} C_DIS
LIN {X -70.072,Y 255.546,Z -49.125,A 0.015,B 0.000,C -180.000} C_DIS
LIN {X -63.541,Y 254.564,Z -49.369,A 0.015,B 0.000,C 180.000} C_DIS
LIN {X -60.025,Y 260.155,Z -49.613,A 0.015,B -0.000,C 180.000} C_DIS
LIN {X -63.738,Y 265.616,Z -49.857,A 0.015,B -0.000,C 180.000} C_DIS
LIN {X -70.230,Y 264.403,Z -50.101,A 0.015,B 0.000,C -180.000} C_DIS
LIN {X -71.720,Y 257.969,Z -50.345,A 0.015,B 0.000,C 180.000} C_DIS
LIN {X -66.422,Y 254.026,Z -50.589,A 0.015,B 0.000,C 180.000} C_DIS
LIN {X -60.686,Y 257.299,Z -50.833,A 0.015,B 0.000,C -180.000} C_DIS
LIN {X -61.387,Y 263.866,Z -51.077,A 0.015,B 0.000,C -180.000} C_DIS
LIN {X -67.684,Y 265.856,Z -51.321,A 0.015,B -0.000,C 180.000} C_DIS
LIN {X -72.031,Y 260.883,Z -51.565,A 0.015,B 0.000,C -180.000} C_DIS
LIN {X -69.216,Y 254.909,Z -51.810,A 0.015,B 0.000,C -180.000} C_DIS
LIN {X -62.615,Y 255.093,Z -52.054,A 0.015,B 0.000,C 180.000} C_DIS
LIN {X -60.138,Y 261.215,Z -52.298,A 0.015,B 0.000,C 180.000} C_DIS
LIN {X -64.755,Y 265.938,Z -52.542,A 0.015,B 0.000,C -180.000} C_DIS
LIN {X -70.932,Y 263.600,Z -52.786,A 0.015,B -0.000,C 180.000} C_DIS
LIN {X -71.265,Y 257.004,Z -53.030,A 0.015,B -0.000,C -180.000} C_DIS
LIN {X -65.356,Y 254.056,Z -53.274,A 0.015,B 0.000,C -180.000} C_DIS
LIN {X -60.286,Y 258.288,Z -53.518,A 0.015,B 0.000,C -180.000} C_DIS
LIN {X -62.133,Y 264.629,Z -53.762,A 0.015,B 0.000,C 180.000} C_DIS
LIN {X -68.682,Y 265.478,Z -54.006,A 0.015,B -0.000,C 180.000} C_DIS
LIN {X -72.085,Y 259.818,Z -54.250,A 0.015,B 0.000,C 180.000} C_DIS
LIN {X -68.262,Y 254.432,Z -54.494,A 0.015,B 0.000,C 180.000} C_DIS
LIN {X -61.796,Y 255.777,Z -54.738,A 0.015,B 0.000,C 180.000} C_DIS
LIN {X -60.436,Y 262.239,Z -54.982,A 0.015,B 0.000,C 180.000} C_DIS
LIN {X -65.813,Y 266.075,Z -55.226,A 0.015,B 0.000,C 180.000} C_DIS
LIN {X -71.481,Y 262.686,Z -55.470,A 0.015,B 0.000,C -180.000} C_DIS
LIN {X -70.648,Y 256.134,Z -55.714,A 0.015,B 0.000,C 180.000} C_DIS
LIN {X -64.311,Y 254.273,Z -55.958,A 0.015,B 0.000,C -180.000} C_DIS
LIN {X -60.066,Y 259.332,Z -56.202,A 0.015,B -0.000,C 180.000} C_DIS
LIN {X -63.001,Y 265.249,Z -56.446,A 0.015,B 0.000,C 180.000} C_DIS
LIN {X -69.598,Y 264.931,Z -56.690,A 0.015,B 0.000,C -180.000} C_DIS
LIN {X -71.950,Y 258.760,Z -56.935,A 0.015,B 0.000,C -180.000} C_DIS
LIN {X -67.239,Y 254.132,Z -57.179,A 0.015,B -0.000,C 180.000} C_DIS
LIN {X -61.110,Y 256.594,Z -57.423,A 0.015,B -0.000,C -180.000} C_DIS
LIN {X -60.910,Y 263.195,Z -57.667,A 0.015,B 0.000,C -180.000} C_DIS
LIN {X -66.878,Y 266.024,Z -57.911,A 0.015,B -0.000,C 180.000} C_DIS
LIN {X -71.861,Y 261.689,Z -58.155,A 0.015,B 0.000,C -180.000} C_DIS
LIN {X -69.887,Y 255.387,Z -58.399,A 0.015,B -0.000,C -180.000} C_DIS
LIN {X -63.322,Y 254.670,Z -58.643,A 0.015,B 0.000,C -180.000} C_DIS
LIN {X -60.034,Y 260.398,Z -58.887,A 0.015,B -0.000,C -180.000} C_DIS
LIN {X -63.965,Y 265.706,Z -59.131,A 0.015,B 0.000,C -180.000} C_DIS
LIN {X -70.402,Y 264.231,Z -59.375,A 0.015,B 0.000,C -180.000} C_DIS
LIN {X -71.631,Y 257.742,Z -59.619,A 0.015,B 0.000,C -180.000} C_DIS
LIN {X -66.178,Y 254.016,Z -59.863,A 0.015,B 0.000,C 180.000} C_DIS
LIN {X -60.579,Y 257.519,Z -60.107,A 0.015,B 0.000,C 180.000} C_DIS
LIN {X -61.545,Y 264.052,Z -60.351,A 0.015,B -0.000,C -180.000} C_DIS
LIN {X -67.918,Y 265.785,Z -60.595,A 0.015,B -0.000,C 180.000} C_DIS
LIN {X -72.060,Y 260.641,Z -60.839,A 0.015,B 0.000,C -180.000} C_DIS
LIN {X -69.006,Y 254.785,Z -61.083,A 0.015,B -0.000,C 180.000} C_DIS
LIN {X -62.417,Y 255.236,Z -61.327,A 0.015,B 0.000,C 180.000} C_DIS
LIN {X -60.190,Y 261.454,Z -61.571,A 0.015,B 0.000,C 180.000} C_DIS
LIN {X -64.994,Y 265.986,Z -61.815,A 0.015,B 0.000,C -180.000} C_DIS
LIN {X -71.071,Y 263.400,Z -62.060,A 0.015,B 0.000,C -180.000} C_DIS
LIN {X -71.138,Y 256.796,Z -62.304,A 0.015,B 0.000,C -180.000} C_DIS
LIN {X -65.114,Y 254.089,Z -62.548,A 0.015,B 0.000,C -180.000} C_DIS
LIN {X -60.220,Y 258.523,Z -62.792,A 0.015,B 0.000,C -180.000} C_DIS
LIN {X -62.321,Y 264.784,Z -63.036,A 0.015,B 0.000,C 180.000} C_DIS
LIN {X -68.899,Y 265.368,Z -63.280,A 0.015,B 0.000,C 180.000} C_DIS
LIN {X -72.070,Y 259.575,Z -63.524,A 0.015,B -0.000,C -180.000} C_DIS
LIN {X -68.033,Y 254.348,Z -63.768,A 0.015,B 0.000,C -180.000} C_DIS
LIN {X -61.627,Y 255.952,Z -64.012,A 0.015,B 0.000,C -180.000} C_DIS
LIN {X -60.529,Y 262.465,Z -64.256,A 0.015,B 0.000,C 180.000} C_DIS
LIN {X -66.057,Y 266.080,Z -64.500,A 0.015,B -0.000,C -180.000} C_DIS
LIN {X -66.452,Y 266.080,Z -64.500,A 0.015,B 0.000,C -180.000} C_DIS
CIRC {X -68.556,Y 265.146,Z -64.500,A 0.015,B 0.000,C 180.000},{X -69.276,Y 262.959,Z -64.500,A 0.015,B 0.000,C 180.000} C_DIS
LIN {X -65.145,Y 221.623,Z -64.500,A 0.015,B 0.000,C 180.000} C_DIS
CIRC {X -63.948,Y 220.592,Z -64.500,A 0.015,B 0.000,C 180.000},{X -62.859,Y 221.737,Z -64.500,A 0.015,B 0.000,C -180.000} C_DIS
LIN {X -62.860,Y 263.241,Z -64.500,A 0.015,B 0.000,C -180.000} C_DIS
CIRC {X -63.692,Y 265.248,Z -64.500,A 0.015,B 0.000,C 180.000},{X -65.699,Y 266.080,Z -64.500,A 0.015,B 0.000,C -180.000} C_DIS
LIN {X -66.057,Y 266.080,Z -64.500,A 0.015,B -0.000,C -180.000} C_DIS
CIRC {X -68.335,Y 266.910,Z -64.500,A 0.015,B 0.000,C -180.000},{X -69.546,Y 269.011,Z -64.500,A 0.015,B 0.000,C -180.000} C_DIS
CIRC {X -71.226,Y 271.030,Z -64.500,A 0.015,B 0.000,C -180.000},{X -73.817,Y 270.602,Z -64.500,A 0.015,B -0.000,C 180.000} C_DIS
CIRC {X -74.816,Y 269.261,Z -64.500,A 0.015,B 0.000,C -180.000},{X -75.060,Y 267.608,Z -64.500,A 0.015,B -0.000,C -180.000} C_DIS
LIN {X -66.905,Y 186.005,Z -64.500,A 0.015,B 0.000,C -180.000} C_DIS
CIRC {X -66.414,Y 184.481,Z -64.500,A 0.015,B 0.000,C 180.000},{X -65.339,Y 183.293,Z -64.500,A 0.015,B 0.000,C 180.000} C_DIS
LIN {X -60.808,Y 180.037,Z -64.500,A 0.015,B -0.000,C 180.000} C_DIS
CIRC {X -58.678,Y 179.877,Z -64.500,A 0.015,B -0.000,C -180.000},{X -57.565,Y 181.700,Z -64.500,A 0.015,B 0.000,C 180.000} C_DIS
LIN {X -57.567,Y 267.520,Z -64.500,A 0.015,B 0.000,C -180.000} C_DIS
CIRC {X -58.696,Y 270.244,Z -64.500,A 0.015,B -0.000,C 180.000},{X -61.420,Y 271.373,Z -64.500,A 0.015,B -0.000,C 180.000} C_DIS
LIN {X -71.653,Y 271.373,Z -64.500,A 0.015,B -0.000,C 180.000} C_DIS
CIRC {X -72.802,Y 271.174,Z -64.500,A 0.015,B 0.000,C -180.000},{X -73.817,Y 270.602,Z -64.500,A 0.015,B 0.000,C -180.000} C_DIS
CIRC {X -76.252,Y 269.154,Z -64.500,A 0.015,B -0.000,C 180.000},{X -79.002,Y 268.477,Z -64.500,A 0.015,B 0.000,C -180.000} C_DIS
CIRC {X -81.682,Y 267.055,Z -64.500,A 0.015,B 0.000,C 180.000},{X -82.563,Y 264.151,Z -64.500,A 0.015,B 0.000,C -180.000} C_DIS
LIN {X -74.700,Y 185.471,Z -64.500,A 0.015,B -0.000,C 180.000} C_DIS
CIRC {X -73.131,Y 180.602,Z -64.500,A 0.015,B 0.000,C 180.000},{X -69.699,Y 176.809,Z -64.500,A 0.015,B 0.000,C -180.000} C_DIS
LIN {X -52.998,Y 164.806,Z -64.500,A 0.015,B 0.000,C -180.000} C_DIS
CIRC {X -50.868,Y 164.647,Z -64.500,A 0.015,B 0.000,C 180.000},{X -49.755,Y 166.469,Z -64.500,A 0.015,B -0.000,C 180.000} C_DIS
LIN {X -49.758,Y 275.330,Z -64.500,A 0.015,B 0.000,C 180.000} C_DIS
CIRC {X -50.887,Y 278.054,Z -64.500,A 0.015,B -0.000,C -180.000},{X -53.611,Y 279.183,Z -64.500,A 0.015,B 0.000,C 180.000} C_DIS
LIN {X -80.282,Y 279.182,Z -64.500,A 0.015,B 0.000,C -180.000} C_DIS
CIRC {X -82.821,Y 278.056,Z -64.500,A 0.015,B 0.000,C 180.000},{X -83.689,Y 275.418,Z -64.500,A 0.015,B 0.000,C -180.000} C_DIS
LIN {X -82.563,Y 264.151,Z -64.500,A 0.015,B 0.000,C 180.000} C_DIS
CIRC {X -83.274,Y 260.543,Z -64.500,A 0.015,B 0.000,C -180.000},{X -85.866,Y 257.935,Z -64.500,A 0.015,B -0.000,C 180.000} C_DIS
CIRC {X -88.459,Y 255.326,Z -64.500,A 0.015,B -0.000,C -180.000},{X -89.169,Y 251.718,Z -64.500,A 0.015,B 0.000,C -180.000} C_DIS
LIN {X -82.153,Y 181.514,Z -64.500,A 0.015,B 0.000,C 180.000} C_DIS
CIRC {X -80.491,Y 176.353,Z -64.500,A 0.015,B 0.000,C 180.000},{X -76.852,Y 172.333,Z -64.500,A 0.015,B 0.000,C -180.000} C_DIS
LIN {X -45.188,Y 149.576,Z -64.500,A 0.015,B 0.000,C 180.000} C_DIS
CIRC {X -43.058,Y 149.416,Z -64.500,A 0.015,B 0.000,C 180.000},{X -41.945,Y 151.239,Z -64.500,A 0.015,B 0.000,C -180.000} C_DIS
LIN {X -41.948,Y 283.140,Z -64.500,A 0.015,B -0.000,C 180.000} C_DIS
CIRC {X -43.077,Y 285.864,Z -64.500,A 0.015,B 0.000,C 180.000},{X -45.802,Y 286.993,Z -64.500,A 0.015,B -0.000,C 180.000} C_DIS
LIN {X -88.911,Y 286.991,Z -64.500,A 0.015,B -0.000,C 180.000} C_DIS
CIRC {X -91.450,Y 285.865,Z -64.500,A 0.015,B 0.000,C 180.000},{X -92.318,Y 283.227,Z -64.500,A 0.015,B 0.000,C -180.000} C_DIS
LIN {X -89.169,Y 251.718,Z -64.500,A 0.015,B -0.000,C 180.000} C_DIS
CIRC {X -89.880,Y 248.110,Z -64.500,A 0.015,B -0.000,C -180.000},{X -92.472,Y 245.502,Z -64.500,A 0.015,B 0.000,C -180.000} C_DIS
CIRC {X -95.065,Y 242.893,Z -64.500,A 0.015,B 0.000,C 180.000},{X -95.775,Y 239.285,Z -64.500,A 0.015,B 0.000,C 180.000} C_DIS
LIN {X -89.573,Y 177.229,Z -64.500,A 0.015,B 0.000,C 180.000} C_DIS
CIRC {X -87.911,Y 172.069,Z -64.500,A 0.015,B -0.000,C -180.000},{X -84.273,Y 168.049,Z -64.500,A 0.015,B 0.000,C 180.000} C_DIS
LIN {X -37.378,Y 134.345,Z -64.500,A 0.015,B -0.000,C -180.000} C_DIS
CIRC {X -35.248,Y 134.186,Z -64.500,A 0.015,B -0.000,C 180.000},{X -34.135,Y 136.008,Z -64.500,A 0.015,B 0.000,C 180.000} C_DIS
LIN {X -34.139,Y 290.949,Z -64.500,A 0.015,B -0.000,C -180.000} C_DIS
CIRC {X -35.268,Y 293.674,Z -64.500,A 0.015,B 0.000,C 180.000},{X -37.992,Y 294.802,Z -64.500,A 0.015,B 0.000,C -180.000} C_DIS
LIN {X -97.541,Y 294.801,Z -64.500,A 0.015,B 0.000,C 180.000} C_DIS
CIRC {X -100.079,Y 293.674,Z -64.500,A 0.015,B 0.000,C 180.000},{X -100.947,Y 291.037,Z -64.500,A 0.015,B 0.000,C 180.000} C_DIS
LIN {X -95.775,Y 239.285,Z -64.500,A 0.015,B 0.000,C 180.000} C_DIS
CIRC {X -96.486,Y 235.677,Z -64.500,A 0.015,B 0.000,C 180.000},{X -99.078,Y 233.069,Z -64.500,A 0.015,B 0.000,C 180.000} C_DIS
CIRC {X -101.671,Y 230.460,Z -64.500,A 0.015,B -0.000,C -180.000},{X -102.381,Y 226.852,Z -64.500,A 0.015,B 0.000,C 180.000} C_DIS
LIN {X -96.994,Y 172.945,Z -64.500,A 0.015,B 0.000,C 180.000} C_DIS
CIRC {X -95.331,Y 167.784,Z -64.500,A 0.015,B -0.000,C -180.000},{X -91.693,Y 163.765,Z -64.500,A 0.015,B 0.000,C 180.000} C_DIS
LIN {X -29.567,Y 119.115,Z -64.500,A 0.015,B 0.000,C 180.000} C_DIS
CIRC {X -27.438,Y 118.956,Z -64.500,A 0.015,B 0.000,C 180.000},{X -26.325,Y 120.778,Z -64.500,A 0.015,B 0.000,C -180.000} C_DIS
LIN {X -26.330,Y 298.759,Z -64.500,A 0.015,B 0.000,C -180.000} C_DIS
CIRC {X -27.458,Y 301.484,Z -64.500,A 0.015,B -0.000,C 180.000},{X -30.183,Y 302.612,Z -64.500,A 0.015,B 0.000,C 180.000} C_DIS
LIN {X -106.170,Y 302.610,Z -64.500,A 0.015,B -0.000,C 180.000} C_DIS
CIRC {X -108.708,Y 301.484,Z -64.500,A 0.015,B 0.000,C 180.000},{X -109.576,Y 298.846,Z -64.500,A 0.015,B 0.000,C 180.000} C_DIS
LIN {X -102.381,Y 226.852,Z -64.500,A 0.015,B -0.000,C -180.000} C_DIS
CIRC {X -103.088,Y 223.271,Z -64.500,A 0.015,B 0.000,C 180.000},{X -105.664,Y 220.685,Z -64.500,A 0.015,B 0.000,C 180.000} C_DIS
CIRC {X -108.238,Y 218.098,Z -64.500,A 0.015,B 0.000,C 180.000},{X -108.947,Y 214.517,Z -64.500,A 0.015,B 0.000,C -180.000} C_DIS
LIN {X -104.325,Y 167.774,Z -64.500,A 0.015,B 0.000,C 180.000} C_DIS
CIRC {X -102.918,Y 163.404,Z -64.500,A 0.015,B 0.000,C 180.000},{X -99.837,Y 160.000,Z -64.500,A 0.015,B 0.000,C -180.000} C_DIS
LIN {X -21.757,Y 103.884,Z -64.500,A 0.015,B -0.000,C 180.000} C_DIS
CIRC {X -19.628,Y 103.725,Z -64.500,A 0.015,B 0.000,C -180.000},{X -18.515,Y 105.547,Z -64.500,A 0.015,B 0.000,C -180.000} C_DIS
LIN {X -18.520,Y 306.569,Z -64.500,A 0.015,B 0.000,C -180.000} C_DIS
CIRC {X -19.649,Y 309.294,Z -64.500,A 0.015,B -0.000,C 180.000},{X -22.373,Y 310.422,Z -64.500,A 0.015,B 0.000,C 180.000} C_DIS
LIN {X -115.319,Y 310.420,Z -64.500,A 0.015,B -0.000,C 180.000} C_DIS
CIRC {X -117.676,Y 309.337,Z -64.500,A 0.015,B 0.000,C 180.000},{X -118.389,Y 306.843,Z -64.500,A 0.015,B -0.000,C -180.000} C_DIS
CIRC {X -118.198,Y 305.702,Z -64.500,A 0.015,B 0.000,C 180.000},{X -117.976,Y 304.566,Z -64.500,A 0.015,B 0.000,C 180.000} C_DIS
CIRC {X -117.769,Y 303.427,Z -64.500,A 0.015,B -0.000,C 180.000},{X -117.623,Y 302.279,Z -64.500,A 0.015,B 0.000,C 180.000} C_DIS
LIN {X -108.947,Y 214.517,Z -64.500,A 0.015,B -0.000,C -180.000} C_DIS
CIRC {X -109.648,Y 210.981,Z -64.500,A 0.015,B 0.000,C -180.000},{X -112.194,Y 208.429,Z -64.500,A 0.015,B 0.000,C 180.000} C_DIS
CIRC {X -114.739,Y 205.876,Z -64.500,A 0.015,B 0.000,C 180.000},{X -115.442,Y 202.341,Z -64.500,A 0.015,B 0.000,C -180.000} C_DIS
LIN {X -111.862,Y 165.832,Z -64.500,A 0.015,B 0.000,C -180.000} C_DIS
CIRC {X -111.801,Y 164.890,Z -64.500,A 0.015,B 0.000,C -180.000},{X -111.805,Y 163.945,Z -64.500,A 0.015,B -0.000,C -180.000} C_DIS
CIRC {X -111.846,Y 163.002,Z -64.500,A 0.015,B 0.000,C 180.000},{X -111.895,Y 162.060,Z -64.500,A 0.015,B 0.000,C 180.000} C_DIS
CIRC {X -111.079,Y 158.655,Z -64.500,A 0.015,B 0.000,C 180.000},{X -108.530,Y 156.256,Z -64.500,A 0.015,B 0.000,C -180.000} C_DIS
CIRC {X -107.668,Y 155.819,Z -64.500,A 0.015,B 0.000,C -180.000},{X -106.810,Y 155.375,Z -64.500,A 0.015,B -0.000,C 180.000} C_DIS
CIRC {X -105.970,Y 154.897,Z -64.500,A 0.015,B -0.000,C 180.000},{X -105.166,Y 154.361,Z -64.500,A 0.015,B 0.000,C 180.000} C_DIS
LIN {X -13.947,Y 88.654,Z -64.500,A 0.015,B -0.000,C -180.000} C_DIS
CIRC {X -11.818,Y 88.495,Z -64.500,A 0.015,B 0.000,C -180.000},{X -10.705,Y 90.317,Z -64.500,A 0.015,B 0.000,C 180.000} C_DIS
LIN {X -10.711,Y 314.379,Z -64.500,A 0.015,B -0.000,C 180.000} C_DIS
CIRC {X -11.839,Y 317.103,Z -64.500,A 0.015,B 0.000,C -180.000},{X -14.564,Y 318.232,Z -64.500,A 0.015,B -0.000,C 180.000} C_DIS
LIN {X -125.792,Y 318.229,Z -64.500,A 0.015,B 0.000,C 180.000} C_DIS
CIRC {X -127.941,Y 317.150,Z -64.500,A 0.015,B 0.000,C 180.000},{X -128.356,Y 314.781,Z -64.500,A 0.015,B -0.000,C -180.000} C_DIS
CIRC {X -127.457,Y 311.751,Z -64.500,A 0.015,B -0.000,C 180.000},{X -126.579,Y 308.715,Z -64.500,A 0.015,B 0.000,C -180.000} C_DIS
CIRC {X -125.817,Y 305.646,Z -64.500,A 0.015,B 0.000,C 180.000},{X -125.266,Y 302.532,Z -64.500,A 0.015,B 0.000,C 180.000} C_DIS
LIN {X -115.442,Y 202.341,Z -64.500,A 0.015,B 0.000,C 180.000} C_DIS
CIRC {X -116.143,Y 198.815,Z -64.500,A 0.015,B 0.000,C 180.000},{X -118.682,Y 196.270,Z -64.500,A 0.015,B 0.000,C -180.000} C_DIS
CIRC {X -121.220,Y 193.725,Z -64.500,A 0.015,B 0.000,C -180.000},{X -121.921,Y 190.199,Z -64.500,A 0.015,B 0.000,C -180.000} C_DIS
LIN {X -119.456,Y 165.073,Z -64.500,A 0.015,B 0.000,C 180.000} C_DIS
CIRC {X -119.386,Y 162.684,Z -64.500,A 0.015,B 0.000,C 180.000},{X -119.651,Y 160.309,Z -64.500,A 0.015,B 0.000,C 180.000} C_DIS
CIRC {X -120.174,Y 157.981,Z -64.500,A 0.015,B 0.000,C 180.000},{X -120.879,Y 155.702,Z -64.500,A 0.015,B 0.000,C 180.000} C_DIS
CIRC {X -120.676,Y 153.209,Z -64.500,A 0.015,B 0.000,C 180.000},{X -118.680,Y 151.700,Z -64.500,A 0.015,B -0.000,C -180.000} C_DIS
CIRC {X -117.052,Y 151.298,Z -64.500,A 0.015,B -0.000,C 180.000},{X -115.438,Y 150.842,Z -64.500,A 0.015,B 0.000,C 180.000} C_DIS
CIRC {X -113.849,Y 150.299,Z -64.500,A 0.015,B 0.000,C 180.000},{X -112.306,Y 149.641,Z -64.500,A 0.015,B 0.000,C 180.000} C_DIS
CIRC {X -111.614,Y 149.308,Z -64.500,A 0.015,B 0.000,C -180.000},{X -110.928,Y 148.965,Z -64.500,A 0.015,B 0.000,C 180.000} C_DIS
CIRC {X -110.257,Y 148.591,Z -64.500,A 0.015,B -0.000,C 180.000},{X -109.617,Y 148.167,Z -64.500,A 0.015,B -0.000,C -180.000} C_DIS
LIN {X -6.137,Y 73.423,Z -64.500,A 0.015,B 0.000,C 180.000} C_DIS
CIRC {X -4.008,Y 73.264,Z -64.500,A 0.015,B 0.000,C -180.000},{X -2.895,Y 75.086,Z -64.500,A 0.015,B -0.000,C -180.000} C_DIS
LIN {X -2.901,Y 322.189,Z -64.500,A 0.015,B 0.000,C 180.000} C_DIS
CIRC {X -4.030,Y 324.913,Z -64.500,A 0.015,B 0.000,C -180.000},{X -6.754,Y 326.042,Z -64.500,A 0.015,B 0.000,C 180.000} C_DIS
LIN {X -138.536,Y 326.038,Z -64.500,A 0.015,B 0.000,C -180.000} C_DIS
CIRC {X -140.474,Y 324.922,Z -64.500,A 0.015,B -0.000,C -180.000},{X -140.481,Y 322.686,Z -64.500,A 0.015,B 0.000,C 180.000} C_DIS
CIRC {X -138.601,Y 319.298,Z -64.500,A 0.015,B 0.000,C -180.000},{X -136.811,Y 315.861,Z -64.500,A 0.015,B 0.000,C 180.000} C_DIS
CIRC {X -135.281,Y 312.294,Z -64.500,A 0.015,B 0.000,C -180.000},{X -134.205,Y 308.564,Z -64.500,A 0.015,B 0.000,C -180.000} C_DIS
CIRC {X -133.782,Y 306.626,Z -64.500,A 0.015,B 0.000,C 180.000},{X -133.371,Y 304.686,Z -64.500,A 0.015,B 0.000,C -180.000} C_DIS
CIRC {X -133.018,Y 302.734,Z -64.500,A 0.015,B 0.000,C 180.000},{X -132.768,Y 300.765,Z -64.500,A 0.015,B 0.000,C 180.000} C_DIS
LIN {X -121.921,Y 190.199,Z -64.500,A 0.015,B 0.000,C 180.000} C_DIS
LIN {X -121.706,Y 189.609,Z -64.330,A 0.015,B -0.000,C 180.000} C_DIS
LIN {X -121.380,Y 189.281,Z -63.865,A 0.015,B 0.000,C 180.000} C_DIS
LIN {X -121.234,Y 189.194,Z -63.230,A 0.015,B 0.000,C 180.000} C_DIS
$VEL.CP = 1.00000
LIN {X -121.234,Y 189.194,Z 11.000,A 0.015,B -0.000,C -180.000} C_DIS
$VEL.CP = 1.00000
LIN {X -206.449,Y 109.973,Z 11.000,A 0.015,B 0.000,C -180.000} C_DIS
$VEL.CP = 1.00000
LIN {X -206.449,Y 109.973,Z -42.731,A 0.015,B 0.000,C 180.000} C_DIS
$VEL.CP = 0.10000
LIN {X -206.467,Y 109.811,Z -43.353,A 0.015,B 0.000,C -180.000} C_DIS
LIN {X -206.495,Y 109.366,Z -43.816,A 0.015,B 0.000,C 180.000} C_DIS
LIN {X -206.480,Y 108.750,Z -44.000,A 0.015,B 0.000,C 180.000} C_DIS
LIN {X -202.456,Y 103.513,Z -44.244,A 0.015,B 0.000,C 180.000} C_DIS
LIN {X -196.045,Y 105.102,Z -44.488,A 0.015,B 0.000,C -180.000} C_DIS
LIN {X -194.932,Y 111.611,Z -44.732,A 0.015,B 0.000,C 180.000} C_DIS
LIN {X -200.450,Y 115.240,Z -44.976,A 0.015,B 0.000,C -180.000} C_DIS
LIN {X -205.986,Y 111.639,Z -45.220,A 0.015,B 0.000,C 180.000} C_DIS
LIN {X -204.905,Y 105.123,Z -45.464,A 0.015,B 0.000,C 180.000} C_DIS
LIN {X -198.502,Y 103.503,Z -45.708,A 0.015,B 0.000,C -180.000} C_DIS
LIN {X -194.452,Y 108.720,Z -45.952,A 0.015,B 0.000,C -180.000} C_DIS
LIN {X -197.609,Y 114.521,Z -46.196,A 0.015,B 0.000,C -180.000} C_DIS
LIN {X -204.189,Y 113.954,Z -46.440,A 0.015,B 0.000,C -180.000} C_DIS
LIN {X -206.305,Y 107.698,Z -46.685,A 0.015,B 0.000,C -180.000} C_DIS
LIN {X -201.422,Y 103.252,Z -46.929,A 0.015,B 0.000,C 180.000} C_DIS
LIN {X -195.391,Y 105.944,Z -47.173,A 0.015,B -0.000,C -180.000} C_DIS
LIN {X -195.442,Y 112.548,Z -47.417,A 0.015,B 0.000,C 180.000} C_DIS
LIN {X -201.513,Y 115.148,Z -47.661,A 0.015,B -0.000,C 180.000} C_DIS
LIN {X -206.328,Y 110.628,Z -47.905,A 0.015,B 0.000,C -180.000} C_DIS
LIN {X -204.116,Y 104.405,Z -48.149,A 0.015,B -0.000,C 180.000} C_DIS
LIN {X -197.528,Y 103.938,Z -48.393,A 0.015,B 0.000,C 180.000} C_DIS
LIN {X -194.460,Y 109.787,Z -48.637,A 0.015,B 0.000,C -180.000} C_DIS
LIN {X -198.589,Y 114.941,Z -48.881,A 0.015,B 0.000,C -180.000} C_DIS
LIN {X -204.966,Y 113.224,Z -49.125,A 0.015,B -0.000,C -180.000} C_DIS
LIN {X -205.948,Y 106.693,Z -49.369,A 0.015,B 0.000,C 180.000} C_DIS
LIN {X -200.358,Y 103.176,Z -49.613,A 0.015,B 0.000,C 180.000} C_DIS
LIN {X -194.896,Y 106.889,Z -49.857,A 0.015,B 0.000,C 180.000} C_DIS
LIN {X -196.109,Y 113.381,Z -50.101,A 0.015,B 0.000,C -180.000} C_DIS
LIN {X -202.543,Y 114.871,Z -50.345,A 0.015,B 0.000,C 180.000} C_DIS
LIN {X -206.486,Y 109.573,Z -50.589,A 0.015,B 0.000,C 180.000} C_DIS
LIN {X -203.213,Y 103.837,Z -50.833,A 0.015,B 0.000,C -180.000} C_DIS
LIN {X -196.646,Y 104.538,Z -51.077,A 0.015,B -0.000,C 180.000} C_DIS
LIN {X -194.656,Y 110.836,Z -51.321,A 0.015,B 0.000,C 180.000} C_DIS
LIN {X -199.629,Y 115.182,Z -51.565,A 0.015,B 0.000,C 180.000} C_DIS
LIN {X -205.603,Y 112.368,Z -51.810,A 0.015,B 0.000,C -180.000} C_DIS
LIN {X -205.419,Y 105.766,Z -52.054,A 0.015,B 0.000,C 180.000} C_DIS
LIN {X -199.297,Y 103.289,Z -52.298,A 0.015,B 0.000,C -180.000} C_DIS
LIN {X -194.575,Y 107.906,Z -52.542,A 0.015,B 0.000,C 180.000} C_DIS
LIN {X -196.912,Y 114.083,Z -52.786,A 0.015,B 0.000,C -180.000} C_DIS
LIN {X -203.508,Y 114.417,Z -53.030,A 0.015,B 0.000,C 180.000} C_DIS
LIN {X -206.457,Y 108.507,Z -53.274,A 0.015,B 0.000,C 180.000} C_DIS
LIN {X -202.224,Y 103.437,Z -53.518,A 0.015,B 0.000,C 180.000} C_DIS
LIN {X -195.883,Y 105.284,Z -53.762,A 0.015,B 0.000,C 180.000} C_DIS
LIN {X -195.034,Y 111.833,Z -54.006,A 0.015,B -0.000,C 180.000} C_DIS
LIN {X -200.694,Y 115.236,Z -54.250,A 0.015,B 0.000,C 180.000} C_DIS
LIN {X -206.080,Y 111.413,Z -54.494,A 0.015,B 0.000,C 180.000} C_DIS
LIN {X -204.736,Y 104.947,Z -54.738,A 0.015,B -0.000,C -180.000} C_DIS
LIN {X -198.273,Y 103.588,Z -54.982,A 0.015,B 0.000,C 180.000} C_DIS
LIN {X -194.437,Y 108.964,Z -55.226,A 0.015,B 0.000,C 180.000} C_DIS
LIN {X -197.826,Y 114.632,Z -55.470,A 0.015,B 0.000,C 180.000} C_DIS
LIN {X -204.378,Y 113.799,Z -55.714,A 0.015,B 0.000,C 180.000} C_DIS
LIN {X -206.240,Y 107.463,Z -55.958,A 0.015,B 0.000,C 180.000} C_DIS
LIN {X -201.180,Y 103.218,Z -56.202,A 0.015,B -0.000,C 180.000} C_DIS
LIN {X -195.264,Y 106.152,Z -56.446,A 0.015,B 0.000,C -180.000} C_DIS
LIN {X -195.581,Y 112.749,Z -56.690,A 0.015,B -0.000,C 180.000} C_DIS
LIN {X -201.752,Y 115.101,Z -56.935,A 0.015,B 0.000,C 180.000} C_DIS
LIN {X -206.380,Y 110.390,Z -57.179,A 0.015,B 0.000,C 180.000} C_DIS
LIN {X -203.919,Y 104.262,Z -57.423,A 0.015,B 0.000,C -180.000} C_DIS
LIN {X -197.317,Y 104.061,Z -57.667,A 0.015,B 0.000,C -180.000} C_DIS
LIN {X -194.489,Y 110.029,Z -57.911,A 0.015,B 0.000,C -180.000} C_DIS
LIN {X -198.823,Y 115.012,Z -58.155,A 0.015,B 0.000,C 180.000} C_DIS
LIN {X -205.125,Y 113.038,Z -58.399,A 0.015,B -0.000,C 180.000} C_DIS
LIN {X -205.842,Y 106.473,Z -58.643,A 0.015,B 0.000,C 180.000} C_DIS
LIN {X -200.114,Y 103.185,Z -58.887,A 0.015,B 0.000,C 180.000} C_DIS
LIN {X -194.807,Y 107.116,Z -59.131,A 0.015,B 0.000,C -180.000} C_DIS
LIN {X -196.281,Y 113.554,Z -59.375,A 0.015,B 0.000,C -180.000} C_DIS
LIN {X -202.770,Y 114.782,Z -59.619,A 0.015,B 0.000,C 180.000} C_DIS
LIN {X -206.496,Y 109.330,Z -59.863,A 0.015,B 0.000,C 180.000} C_DIS
LIN {X -202.994,Y 103.731,Z -60.107,A 0.015,B 0.000,C -180.000} C_DIS
LIN {X -196.460,Y 104.696,Z -60.351,A 0.015,B 0.000,C 180.000} C_DIS
LIN {X -194.727,Y 111.069,Z -60.595,A 0.015,B 0.000,C 180.000} C_DIS
LIN {X -199.871,Y 115.211,Z -60.839,A 0.015,B 0.000,C 180.000} C_DIS
LIN {X -205.727,Y 112.158,Z -61.083,A 0.015,B 0.000,C 180.000} C_DIS
LIN {X -205.276,Y 105.569,Z -61.327,A 0.015,B 0.000,C -180.000} C_DIS
LIN {X -199.059,Y 103.341,Z -61.571,A 0.015,B 0.000,C 180.000} C_DIS
LIN {X -194.527,Y 108.145,Z -61.815,A 0.015,B 0.000,C 180.000} C_DIS
LIN {X -197.112,Y 114.223,Z -62.060,A 0.015,B -0.000,C 180.000} C_DIS
LIN {X -203.716,Y 114.289,Z -62.304,A 0.015,B 0.000,C 180.000} C_DIS
LIN {X -206.423,Y 108.265,Z -62.548,A 0.015,B -0.000,C -180.000} C_DIS
LIN {X -201.989,Y 103.371,Z -62.792,A 0.015,B 0.000,C -180.000} C_DIS
LIN {X -195.728,Y 105.472,Z -63.036,A 0.015,B 0.000,C 180.000} C_DIS
LIN {X -195.144,Y 112.051,Z -63.280,A 0.015,B 0.000,C 180.000} C_DIS
LIN {X -200.937,Y 115.222,Z -63.524,A 0.015,B 0.000,C 180.000} C_DIS
LIN {X -206.164,Y 111.185,Z -63.768,A 0.015,B 0.000,C -180.000} C_DIS
LIN {X -204.560,Y 104.778,Z -64.012,A 0.015,B 0.000,C 180.000} C_DIS
LIN {X -198.048,Y 103.681,Z -64.256,A 0.015,B 0.000,C 180.000} C_DIS
LIN {X -194.432,Y 109.208,Z -64.500,A 0.015,B 0.000,C 180.000} C_DIS
CIRC {X -196.756,Y 111.531,Z -64.500,A 0.015,B 0.000,C 180.000},{X -199.080,Y 109.208,Z -64.500,A 0.015,B 0.000,C 180.000} C_DIS
CIRC {X -196.756,Y 106.884,Z -64.500,A 0.015,B 0.000,C 180.000},{X -194.432,Y 109.208,Z -64.500,A 0.015,B 0.000,C -180.000} C_DIS
CIRC {X -193.872,Y 111.256,Z -64.500,A 0.015,B 0.000,C 180.000},{X -192.347,Y 112.733,Z -64.500,A 0.015,B 0.000,C -180.000} C_DIS
CIRC {X -191.132,Y 114.776,Z -64.500,A 0.015,B -0.000,C -180.000},{X -192.330,Y 116.829,Z -64.500,A 0.015,B -0.000,C -180.000} C_DIS
CIRC {X -193.084,Y 117.278,Z -64.500,A 0.015,B 0.000,C -180.000},{X -193.814,Y 117.764,Z -64.500,A 0.015,B 0.000,C -180.000} C_DIS
CIRC {X -196.756,Y 118.696,Z -64.500,A 0.015,B -0.000,C -180.000},{X -199.698,Y 117.764,Z -64.500,A 0.015,B 0.000,C 180.000} C_DIS
CIRC {X -201.103,Y 116.874,Z -64.500,A 0.015,B 0.000,C 180.000},{X -202.588,Y 116.125,Z -64.500,A 0.015,B 0.000,C 180.000} C_DIS
CIRC {X -204.950,Y 114.014,Z -64.500,A 0.015,B -0.000,C -180.000},{X -205.637,Y 110.922,Z -64.500,A 0.015,B 0.000,C 180.000} C_DIS
CIRC {X -205.565,Y 109.268,Z -64.500,A 0.015,B 0.000,C -180.000},{X -205.653,Y 107.615,Z -64.500,A 0.015,B 0.000,C -180.000} C_DIS
CIRC {X -204.998,Y 104.512,Z -64.500,A 0.015,B -0.000,C 180.000},{X -202.663,Y 102.367,Z -64.500,A 0.015,B 0.000,C -180.000} C_DIS
CIRC {X -201.227,Y 101.618,Z -64.500,A 0.015,B 0.000,C -180.000},{X -199.869,Y 100.736,Z -64.500,A 0.015,B -0.000,C 180.000} C_DIS
CIRC {X -196.859,Y 99.736,Z -64.500,A 0.015,B 0.000,C 180.000},{X -193.814,Y 100.624,Z -64.500,A 0.015,B 0.000,C -180.000} C_DIS
CIRC {X -193.079,Y 101.102,Z -64.500,A 0.015,B -0.000,C -180.000},{X -192.334,Y 101.564,Z -64.500,A 0.015,B 0.000,C 180.000} C_DIS
CIRC {X -191.573,Y 101.999,Z -64.500,A 0.015,B 0.000,C 180.000},{X -190.791,Y 102.395,Z -64.500,A 0.015,B 0.000,C 180.000} C_DIS
CIRC {X -188.498,Y 104.537,Z -64.500,A 0.015,B 0.000,C -180.000},{X -187.859,Y 107.610,Z -64.500,A 0.015,B 0.000,C -180.000} C_DIS
CIRC {X -187.947,Y 109.266,Z -64.500,A 0.015,B 0.000,C -180.000},{X -187.875,Y 110.922,Z -64.500,A 0.015,B -0.000,C -180.000} C_DIS
CIRC {X -188.562,Y 114.014,Z -64.500,A 0.015,B 0.000,C 180.000},{X -190.924,Y 116.125,Z -64.500,A 0.015,B 0.000,C 180.000} C_DIS
CIRC {X -191.635,Y 116.461,Z -64.500,A 0.015,B -0.000,C -180.000},{X -192.330,Y 116.829,Z -64.500,A 0.015,B 0.000,C 180.000} C_DIS
LIN {X -192.937,Y 116.991,Z -64.330,A 0.015,B 0.000,C -180.000} C_DIS
LIN {X -193.393,Y 116.912,Z -63.865,A 0.015,B 0.000,C 180.000} C_DIS
LIN {X -193.548,Y 116.842,Z -63.230,A 0.015,B 0.000,C -180.000} C_DIS
$VEL.CP = 1.00000
LIN {X -193.548,Y 116.842,Z 11.000,A 0.015,B 0.000,C 180.000} C_DIS
$VEL.CP = 1.00000
LIN {X -195.986,Y 9.514,Z 11.000,A 0.015,B 0.000,C 180.000} C_DIS
$VEL.CP = 1.00000
LIN {X -195.986,Y 9.514,Z -42.731,A 0.015,B 0.000,C -180.000} C_DIS
$VEL.CP = 0.10000
LIN {X -196.148,Y 9.532,Z -43.353,A 0.015,B -0.000,C 180.000} C_DIS
LIN {X -196.594,Y 9.561,Z -43.816,A 0.015,B 0.000,C 180.000} C_DIS
LIN {X -197.210,Y 9.545,Z -44.000,A 0.015,B 0.000,C 180.000} C_DIS
LIN {X -202.446,Y 5.521,Z -44.244,A 0.015,B 0.000,C 180.000} C_DIS
LIN {X -200.858,Y -0.889,Z -44.488,A 0.015,B 0.000,C 180.000} C_DIS
LIN {X -194.348,Y -2.003,Z -44.732,A 0.015,B 0.000,C 180.000} C_DIS
LIN {X -190.719,Y 3.515,Z -44.976,A 0.015,B 0.000,C -180.000} C_DIS
LIN {X -194.321,Y 9.051,Z -45.220,A 0.015,B 0.000,C 180.000} C_DIS
LIN {X -200.836,Y 7.970,Z -45.464,A 0.015,B -0.000,C 180.000} C_DIS
LIN {X -202.456,Y 1.567,Z -45.708,A 0.015,B 0.000,C 180.000} C_DIS
LIN {X -197.239,Y -2.483,Z -45.952,A 0.015,B 0.000,C -180.000} C_DIS
LIN {X -191.438,Y 0.674,Z -46.196,A 0.015,B 0.000,C 180.000} C_DIS
LIN {X -192.006,Y 7.254,Z -46.440,A 0.015,B 0.000,C -180.000} C_DIS
LIN {X -198.262,Y 9.371,Z -46.685,A 0.015,B 0.000,C -180.000} C_DIS
LIN {X -202.708,Y 4.487,Z -46.929,A 0.015,B 0.000,C 180.000} C_DIS
LIN {X -200.015,Y -1.543,Z -47.173,A 0.015,B 0.000,C 180.000} C_DIS
LIN {X -193.411,Y -1.493,Z -47.417,A 0.015,B 0.000,C -180.000} C_DIS
LIN {X -190.811,Y 4.578,Z -47.661,A 0.015,B 0.000,C 180.000} C_DIS
LIN {X -195.331,Y 9.393,Z -47.905,A 0.015,B 0.000,C -180.000} C_DIS
LIN {X -201.554,Y 7.181,Z -48.149,A 0.015,B -0.000,C 180.000} C_DIS
LIN {X -202.021,Y 0.593,Z -48.393,A 0.015,B -0.000,C -180.000} C_DIS
LIN {X -196.172,Y -2.474,Z -48.637,A 0.015,B -0.000,C -180.000} C_DIS
LIN {X -191.018,Y 1.655,Z -48.881,A 0.015,B 0.000,C 180.000} C_DIS
LIN {X -192.736,Y 8.032,Z -49.125,A 0.015,B 0.000,C -180.000} C_DIS
LIN {X -199.267,Y 9.013,Z -49.369,A 0.015,B 0.000,C 180.000} C_DIS
LIN {X -202.783,Y 3.423,Z -49.613,A 0.015,B -0.000,C -180.000} C_DIS
LIN {X -199.071,Y -2.039,Z -49.857,A 0.015,B 0.000,C 180.000} C_DIS
LIN {X -192.579,Y -0.826,Z -50.101,A 0.015,B 0.000,C 180.000} C_DIS
LIN {X -191.088,Y 5.608,Z -50.345,A 0.015,B 0.000,C -180.000} C_DIS
LIN {X -196.386,Y 9.552,Z -50.589,A 0.015,B 0.000,C -180.000} C_DIS
LIN {X -202.122,Y 6.278,Z -50.833,A 0.015,B 0.000,C 180.000} C_DIS
LIN {X -201.421,Y -0.289,Z -51.077,A 0.015,B -0.000,C 180.000} C_DIS
LIN {X -195.124,Y -2.279,Z -51.321,A 0.015,B 0.000,C 180.000} C_DIS
LIN {X -190.778,Y 2.694,Z -51.565,A 0.015,B 0.000,C 180.000} C_DIS
LIN {X -193.592,Y 8.669,Z -51.810,A 0.015,B 0.000,C 180.000} C_DIS
LIN {X -200.193,Y 8.485,Z -52.054,A 0.015,B -0.000,C -180.000} C_DIS
LIN {X -202.670,Y 2.362,Z -52.298,A 0.015,B 0.000,C -180.000} C_DIS
LIN {X -198.053,Y -2.360,Z -52.542,A 0.015,B 0.000,C 180.000} C_DIS
LIN {X -191.877,Y -0.023,Z -52.786,A 0.015,B 0.000,C 180.000} C_DIS
LIN {X -191.543,Y 6.573,Z -53.030,A 0.015,B 0.000,C 180.000} C_DIS
LIN {X -197.452,Y 9.522,Z -53.274,A 0.015,B 0.000,C 180.000} C_DIS
LIN {X -202.522,Y 5.289,Z -53.518,A 0.015,B -0.000,C 180.000} C_DIS
LIN {X -200.676,Y -1.052,Z -53.762,A 0.015,B -0.000,C 180.000} C_DIS
LIN {X -194.126,Y -1.901,Z -54.006,A 0.015,B -0.000,C 180.000} C_DIS
LIN {X -190.724,Y 3.759,Z -54.250,A 0.015,B 0.000,C -180.000} C_DIS
LIN {X -194.546,Y 9.145,Z -54.494,A 0.015,B 0.000,C -180.000} C_DIS
LIN {X -201.012,Y 7.801,Z -54.738,A 0.015,B -0.000,C 180.000} C_DIS
LIN {X -202.372,Y 1.338,Z -54.982,A 0.015,B 0.000,C -180.000} C_DIS
LIN {X -196.996,Y -2.497,Z -55.226,A 0.015,B -0.000,C -180.000} C_DIS
LIN {X -191.327,Y 0.891,Z -55.470,A 0.015,B 0.000,C 180.000} C_DIS
LIN {X -192.160,Y 7.443,Z -55.714,A 0.015,B -0.000,C -180.000} C_DIS
LIN {X -198.497,Y 9.305,Z -55.958,A 0.015,B 0.000,C -180.000} C_DIS
LIN {X -202.742,Y 4.245,Z -56.202,A 0.015,B 0.000,C 180.000} C_DIS
LIN {X -199.807,Y -1.671,Z -56.446,A 0.015,B 0.000,C 180.000} C_DIS
LIN {X -193.211,Y -1.354,Z -56.690,A 0.015,B 0.000,C 180.000} C_DIS
LIN {X -190.858,Y 4.817,Z -56.935,A 0.015,B 0.000,C -180.000} C_DIS
LIN {X -195.569,Y 9.446,Z -57.179,A 0.015,B 0.000,C 180.000} C_DIS
LIN {X -201.698,Y 6.984,Z -57.423,A 0.015,B -0.000,C 180.000} C_DIS
LIN {X -201.898,Y 0.383,Z -57.667,A 0.015,B 0.000,C -180.000} C_DIS
LIN {X -195.930,Y -2.446,Z -57.911,A 0.015,B 0.000,C 180.000} C_DIS
LIN {X -190.947,Y 1.888,Z -58.155,A 0.015,B -0.000,C 180.000} C_DIS
LIN {X -192.921,Y 8.190,Z -58.399,A 0.015,B -0.000,C -180.000} C_DIS
LIN {X -199.486,Y 8.907,Z -58.643,A 0.015,B 0.000,C 180.000} C_DIS
LIN {X -202.774,Y 3.179,Z -58.887,A 0.015,B 0.000,C -180.000} C_DIS
LIN {X -198.844,Y -2.128,Z -59.131,A 0.015,B 0.000,C -180.000} C_DIS
LIN {X -192.406,Y -0.654,Z -59.375,A 0.015,B 0.000,C 180.000} C_DIS
LIN {X -191.177,Y 5.835,Z -59.619,A 0.015,B 0.000,C -180.000} C_DIS
LIN {X -196.630,Y 9.561,Z -59.863,A 0.015,B -0.000,C 180.000} C_DIS
LIN {X -202.229,Y 6.059,Z -60.107,A 0.015,B 0.000,C 180.000} C_DIS
LIN {X -201.263,Y -0.475,Z -60.351,A 0.015,B 0.000,C 180.000} C_DIS
LIN {X -194.890,Y -2.208,Z -60.595,A 0.015,B 0.000,C 180.000} C_DIS
LIN {X -190.749,Y 2.936,Z -60.839,A 0.015,B 0.000,C 180.000} C_DIS
LIN {X -193.802,Y 8.792,Z -61.083,A 0.015,B -0.000,C 180.000} C_DIS
LIN {X -200.391,Y 8.341,Z -61.327,A 0.015,B 0.000,C 180.000} C_DIS
LIN {X -202.618,Y 2.124,Z -61.571,A 0.015,B 0.000,C 180.000} C_DIS
LIN {X -197.814,Y -2.408,Z -61.815,A 0.015,B 0.000,C -180.000} C_DIS
LIN {X -191.737,Y 0.177,Z -62.060,A 0.015,B -0.000,C -180.000} C_DIS
LIN {X -191.670,Y 6.781,Z -62.304,A 0.015,B 0.000,C 180.000} C_DIS
LIN {X -197.694,Y 9.489,Z -62.548,A 0.015,B 0.000,C -180.000} C_DIS
LIN {X -202.588,Y 5.055,Z -62.792,A 0.015,B -0.000,C 180.000} C_DIS
LIN {X -200.487,Y -1.207,Z -63.036,A 0.015,B 0.000,C -180.000} C_DIS
LIN {X -193.909,Y -1.790,Z -63.280,A 0.015,B -0.000,C 180.000} C_DIS
LIN {X -190.738,Y 4.003,Z -63.524,A 0.015,B 0.000,C 180.000} C_DIS
LIN {X -194.775,Y 9.230,Z -63.768,A 0.015,B 0.000,C -180.000} C_DIS
LIN {X -201.181,Y 7.625,Z -64.012,A 0.015,B 0.000,C 180.000} C_DIS
LIN {X -202.279,Y 1.113,Z -64.256,A 0.015,B 0.000,C -180.000} C_DIS
LIN {X -196.752,Y -2.502,Z -64.500,A 0.015,B 0.000,C -180.000} C_DIS
LIN {X -193.372,Y -2.502,Z -64.500,A 0.015,B 0.000,C 180.000} C_DIS
CIRC {X -192.012,Y -1.404,Z -64.500,A 0.015,B 0.000,C -180.000},{X -192.799,Y 0.157,Z -64.500,A 0.015,B 0.000,C -180.000} C_DIS
CIRC {X -193.541,Y 0.498,Z -64.500,A 0.015,B 0.000,C -180.000},{X -194.278,Y 0.848,Z -64.500,A 0.015,B 0.000,C 180.000} C_DIS
CIRC {X -195.008,Y 1.213,Z -64.500,A 0.015,B 0.000,C 180.000},{X -195.727,Y 1.598,Z -64.500,A 0.015,B 0.000,C -180.000} C_DIS
CIRC {X -196.760,Y 1.863,Z -64.500,A 0.015,B 0.000,C -180.000},{X -197.791,Y 1.590,Z -64.500,A 0.015,B 0.000,C -180.000} C_DIS
CIRC {X -198.493,Y 1.206,Z -64.500,A 0.015,B 0.000,C -180.000},{X -199.205,Y 0.841,Z -64.500,A 0.015,B -0.000,C 180.000} C_DIS
CIRC {X -199.925,Y 0.493,Z -64.500,A 0.015,B 0.000,C 180.000},{X -200.651,Y 0.157,Z -64.500,A 0.015,B -0.000,C 180.000} C_DIS
CIRC {X -201.439,Y -1.404,Z -64.500,A 0.015,B -0.000,C 180.000},{X -200.079,Y -2.502,Z -64.500,A 0.015,B 0.000,C -180.000} C_DIS
LIN {X -196.752,Y -2.502,Z -64.500,A 0.015,B 0.000,C -180.000} C_DIS
CIRC {X -194.703,Y -3.123,Z -64.500,A 0.015,B 0.000,C -180.000},{X -193.343,Y -4.775,Z -64.500,A 0.015,B 0.000,C -180.000} C_DIS
CIRC {X -191.983,Y -6.427,Z -64.500,A 0.015,B 0.000,C 180.000},{X -189.934,Y -7.047,Z -64.500,A 0.015,B 0.000,C -180.000} C_DIS
LIN {X -172.265,Y -7.047,Z -64.500,A 0.015,B 0.000,C 180.000} C_DIS
CIRC {X -170.905,Y -5.949,Z -64.500,A 0.015,B -0.000,C 180.000},{X -171.692,Y -4.388,Z -64.500,A 0.015,B 0.000,C 180.000} C_DIS
CIRC {X -177.357,Y -1.900,Z -64.500,A 0.015,B 0.000,C 180.000},{X -183.072,Y 0.471,Z -64.500,A 0.015,B 0.000,C -180.000} C_DIS
CIRC {X -188.724,Y 2.998,Z -64.500,A 0.015,B 0.000,C -180.000},{X -194.170,Y 5.943,Z -64.500,A 0.015,B -0.000,C 180.000} C_DIS
CIRC {X -196.778,Y 6.650,Z -64.500,A 0.015,B -0.000,C 180.000},{X -199.381,Y 5.923,Z -64.500,A 0.015,B 0.000,C 180.000} C_DIS
CIRC {X -204.794,Y 2.960,Z -64.500,A 0.015,B 0.000,C 180.000},{X -210.426,Y 0.440,Z -64.500,A 0.015,B -0.000,C 180.000} C_DIS
CIRC {X -216.125,Y -1.913,Z -64.500,A 0.015,B 0.000,C 180.000},{X -221.773,Y -4.388,Z -64.500,A 0.015,B 0.000,C 180.000} C_DIS
